C05466=1030.295,97.763,400.155,168.679,44.365,158.305
C05467=1030.301,98.012,400.136,168.682,44.363,158.304
C05468=1030.307,98.261,400.117,168.684,44.361,158.304
C05469=1030.314,98.510,400.099,168.687,44.358,158.304
C05470=1030.319,98.759,400.079,168.688,44.356,158.304
C05471=1030.326,99.008,400.060,168.691,44.354,158.304
C05472=1030.332,99.258,400.041,168.693,44.353,158.304
C05473=1030.338,99.507,400.022,168.696,44.351,158.303
C05474=1030.344,99.756,400.003,168.698,44.349,158.303
C05475=1030.350,100.005,399.984,168.701,44.347,158.303
C05476=1030.356,100.254,399.964,168.704,44.345,158.303
C05477=1030.362,100.504,399.945,168.706,44.343,158.303
C05478=1030.368,100.754,399.926,168.708,44.341,158.303
C05479=1030.375,101.002,399.906,168.710,44.339,158.303
C05480=1030.381,101.252,399.887,168.713,44.337,158.302
C05481=1030.386,101.501,399.868,168.715,44.335,158.302
C05482=1030.393,101.750,399.848,168.718,44.334,158.302
C05483=1030.399,101.999,399.829,168.721,44.332,158.302
C05484=1030.404,102.249,399.810,168.723,44.330,158.302
C05485=1030.410,102.497,399.790,168.725,44.328,158.302
C05486=1030.417,102.746,399.771,168.727,44.326,158.302
C05487=1030.422,102.996,399.752,168.730,44.324,158.301
C05488=1030.428,103.245,399.732,168.733,44.322,158.301
C05489=1030.435,103.494,399.713,168.735,44.320,158.301
C05490=1030.441,103.743,399.693,168.738,44.318,158.301
C05491=1030.447,103.992,399.674,168.740,44.316,158.301
C05492=1030.453,104.242,399.655,168.742,44.315,158.301
C05493=1030.460,104.491,399.635,168.744,44.313,158.301
C05494=1030.465,104.740,399.616,168.747,44.311,158.300
C05495=1030.471,104.989,399.596,168.749,44.308,158.300
C05496=1030.477,105.238,399.577,168.752,44.306,158.300
C05497=1030.483,105.487,399.558,168.755,44.304,158.300
C05498=1030.489,105.736,399.538,168.757,44.303,158.300
C05499=1030.495,105.986,399.519,168.760,44.301,158.300
C05500=1030.502,106.235,399.499,168.761,44.299,158.299
C05501=1030.508,106.484,399.480,168.764,44.297,158.299
C05502=1030.514,106.733,399.460,168.767,44.295,158.299
C05503=1030.520,106.983,399.441,168.769,44.293,158.299
C05504=1030.526,107.231,399.421,168.772,44.291,158.299
C05505=1030.532,107.481,399.402,168.774,44.289,158.299
C05506=1030.538,107.729,399.382,168.777,44.287,158.299
C05507=1030.546,108.015,399.360,168.779,44.285,158.298
C05508=1030.552,108.300,399.338,168.782,44.283,158.298
C05509=1030.560,108.586,399.315,168.785,44.281,158.298
C05510=1030.566,108.871,399.293,168.788,44.278,158.298
C05511=1030.573,109.120,399.274,168.790,44.276,158.298
C05512=1030.579,109.368,399.254,168.793,44.274,158.298
C05513=1030.585,109.619,399.234,168.796,44.272,158.297
C05514=1030.591,109.867,399.214,168.798,44.271,158.297
C05515=1030.597,110.116,399.195,168.801,44.269,158.297
C05516=1030.603,110.365,399.175,168.803,44.267,158.297
C05517=1030.610,110.615,399.156,168.805,44.265,158.297
C05518=1030.616,110.864,399.136,168.807,44.263,158.297
C05519=1030.622,111.113,399.116,168.810,44.261,158.297
C05520=1030.627,111.362,399.097,168.813,44.259,158.296
C05521=1030.633,111.611,399.077,168.815,44.257,158.296
C05522=1030.640,111.861,399.056,168.818,44.255,158.296
C05523=1030.646,112.110,399.037,168.820,44.253,158.296
C05524=1030.652,112.359,399.017,168.823,44.252,158.296
C05525=1030.658,112.608,398.997,168.826,44.250,158.296
C05526=1030.663,112.857,398.978,168.828,44.248,158.296
C05527=1030.670,113.107,398.958,168.830,44.246,158.295
C05528=1030.676,113.356,398.938,168.832,44.244,158.295
C05529=1030.682,113.604,398.918,168.835,44.242,158.295
C05530=1030.688,113.854,398.898,168.838,44.241,158.295
C05531=1030.694,114.103,398.878,168.840,44.239,158.295
C05532=1030.699,114.352,398.858,168.843,44.237,158.295
C05533=1030.705,114.601,398.838,168.845,44.235,158.295
C05534=1030.711,114.850,398.818,168.847,44.234,158.294
C05535=1030.717,115.099,398.798,168.850,44.232,158.294
C05536=1030.724,115.349,398.778,168.852,44.230,158.294
C05537=1030.729,115.598,398.758,168.855,44.228,158.294
C05538=1030.735,115.847,398.738,168.858,44.227,158.294
C05539=1030.741,116.096,398.718,168.860,44.225,158.294
C05540=1030.748,116.345,398.697,168.863,44.223,158.294
C05541=1030.754,116.594,398.677,168.865,44.221,158.294
C05542=1030.759,116.843,398.657,168.867,44.219,158.293
C05543=1030.765,117.092,398.637,168.870,44.217,158.293
C05544=1030.771,117.342,398.617,168.872,44.215,158.293
C05545=1030.777,117.590,398.597,168.875,44.213,158.293
C05546=1030.783,117.840,398.577,168.878,44.212,158.293
C05547=1030.788,118.089,398.557,168.880,44.210,158.293
C05548=1030.795,118.338,398.536,168.883,44.208,158.293
C05549=1030.801,118.587,398.516,168.885,44.206,158.293
C05550=1030.807,118.836,398.497,168.888,44.204,158.293
C05551=1030.813,119.086,398.476,168.889,44.203,158.292
C05552=1030.819,119.335,398.456,168.892,44.201,158.292
C05553=1030.825,119.584,398.436,168.895,44.199,158.292
C05554=1030.831,119.833,398.415,168.897,44.197,158.292
C05555=1030.837,120.082,398.395,168.900,44.195,158.292
C05556=1030.843,120.331,398.375,168.903,44.194,158.292
C05557=1030.849,120.581,398.355,168.905,44.192,158.292
C05558=1030.855,120.829,398.335,168.908,44.190,158.291
C05559=1030.861,121.078,398.315,168.910,44.188,158.291
C05560=1030.867,121.328,398.294,168.913,44.186,158.291
C05561=1030.873,121.577,398.274,168.916,44.184,158.291
C05562=1030.879,121.826,398.254,168.918,44.182,158.291
C05563=1030.886,122.075,398.233,168.920,44.181,158.291
C05564=1030.892,122.324,398.213,168.922,44.179,158.291
C05565=1030.897,122.573,398.193,168.925,44.177,158.290
C05566=1030.904,122.822,398.172,168.927,44.175,158.290
C05567=1030.910,123.071,398.152,168.930,44.173,158.290
C05568=1030.916,123.320,398.132,168.933,44.172,158.290
C05569=1030.922,123.569,398.111,168.935,44.170,158.290
C05570=1030.928,123.818,398.091,168.938,44.168,158.290
C05571=1030.935,124.104,398.067,168.940,44.165,158.290
C05572=1030.942,124.388,398.045,168.944,44.163,158.290
C05573=1030.949,124.673,398.021,168.947,44.161,158.289
C05574=1030.956,124.959,397.997,168.950,44.159,158.289
C05575=1030.962,125.208,397.977,168.953,44.157,158.289
C05576=1030.968,125.457,397.957,168.955,44.156,158.289
C05577=1030.974,125.706,397.937,168.958,44.154,158.289
C05578=1030.980,125.955,397.917,168.960,44.152,158.289
C05579=1030.986,126.205,397.896,168.962,44.150,158.289
C05580=1030.993,126.453,397.876,168.965,44.148,158.288
C05581=1030.999,126.702,397.855,168.967,44.146,158.288
C05582=1031.004,126.951,397.835,168.970,44.144,158.288
C05583=1031.011,127.201,397.814,168.973,44.142,158.288
C05584=1031.017,127.450,397.794,168.975,44.141,158.288
C05585=1031.024,127.699,397.773,168.978,44.139,158.288
C05586=1031.029,127.948,397.753,168.980,44.137,158.288
C05587=1031.036,128.197,397.733,168.983,44.135,158.287
C05588=1031.042,128.446,397.713,168.985,44.133,158.287
C05589=1031.049,128.695,397.692,168.988,44.131,158.287
C05590=1031.054,128.944,397.671,168.991,44.129,158.287
C05591=1031.060,129.194,397.651,168.993,44.128,158.287
C05592=1031.066,129.442,397.631,168.996,44.126,158.287
C05593=1031.073,129.692,397.609,168.999,44.124,158.287
C05594=1031.079,129.940,397.589,169.001,44.122,158.287
C05595=1031.085,130.190,397.569,169.004,44.120,158.286
C05596=1031.092,130.438,397.548,169.006,44.118,158.286
C05597=1031.097,130.688,397.527,169.009,44.116,158.286
C05598=1031.103,130.937,397.507,169.012,44.115,158.286
C05599=1031.110,131.186,397.486,169.014,44.113,158.286
C05600=1031.115,131.435,397.465,169.017,44.111,158.286
C05601=1031.122,131.684,397.444,169.020,44.110,158.286
C05602=1031.127,131.933,397.423,169.022,44.108,158.286
C05603=1031.134,132.183,397.403,169.025,44.106,158.285
C05604=1031.139,132.431,397.382,169.027,44.104,158.285
C05605=1031.146,132.681,397.362,169.030,44.102,158.285
C05606=1031.151,132.929,397.340,169.033,44.101,158.285
C05607=1031.157,133.179,397.319,169.035,44.099,158.285
C05608=1031.163,133.427,397.299,169.038,44.097,158.285
C05609=1031.169,133.677,397.278,169.041,44.095,158.285
C05610=1031.176,133.925,397.257,169.043,44.093,158.285
C05611=1031.181,134.175,397.236,169.046,44.091,158.284
C05612=1031.187,134.423,397.215,169.049,44.090,158.284
C05613=1031.194,134.673,397.195,169.051,44.088,158.284
C05614=1031.199,134.922,397.173,169.054,44.086,158.284
C05615=1031.206,135.170,397.152,169.056,44.084,158.284
C05616=1031.211,135.420,397.132,169.059,44.082,158.284
C05617=1031.217,135.669,397.110,169.062,44.081,158.284
C05618=1031.224,135.918,397.090,169.064,44.079,158.284
C05619=1031.230,136.167,397.068,169.067,44.077,158.284
C05620=1031.236,136.416,397.048,169.069,44.075,158.283
C05621=1031.242,136.665,397.027,169.072,44.074,158.283
C05622=1031.248,136.914,397.005,169.075,44.072,158.283
C05623=1031.255,137.163,396.985,169.077,44.070,158.283
C05624=1031.260,137.412,396.964,169.080,44.069,158.283
C05625=1031.266,137.661,396.942,169.083,44.067,158.283
C05626=1031.272,137.910,396.922,169.085,44.065,158.283
C05627=1031.278,138.159,396.900,169.088,44.064,158.283
C05628=1031.284,138.408,396.879,169.091,44.062,158.283
C05629=1031.290,138.658,396.858,169.093,44.060,158.282
C05630=1031.297,138.906,396.837,169.096,44.058,158.282
C05631=1031.302,139.155,396.816,169.099,44.057,158.282
C05632=1031.308,139.405,396.795,169.101,44.055,158.282
C05633=1031.314,139.654,396.773,169.104,44.053,158.282
C05634=1031.320,139.902,396.752,169.106,44.051,158.282
C05635=1031.327,140.187,396.728,169.110,44.049,158.282
C05636=1031.334,140.473,396.704,169.113,44.048,158.282
C05637=1031.341,140.758,396.679,169.115,44.046,158.282
C05638=1031.347,141.042,396.655,169.119,44.044,158.282
C05639=1031.354,141.291,396.633,169.122,44.042,158.281
C05640=1031.360,141.541,396.613,169.124,44.040,158.281
C05641=1031.365,141.789,396.591,169.127,44.039,158.281
C05642=1031.371,142.039,396.570,169.130,44.037,158.281
C05643=1031.378,142.287,396.549,169.132,44.035,158.281
C05644=1031.384,142.536,396.527,169.135,44.033,158.281
C05645=1031.390,142.785,396.506,169.138,44.032,158.281
C05646=1031.396,143.034,396.484,169.140,44.030,158.281
C05647=1031.401,143.283,396.463,169.143,44.028,158.281
C05648=1031.407,143.533,396.442,169.146,44.027,158.281
C05649=1031.414,143.782,396.420,169.148,44.025,158.280
C05650=1031.420,144.030,396.400,169.151,44.023,158.280
C05651=1031.426,144.279,396.378,169.153,44.021,158.280
C05652=1031.432,144.528,396.356,169.156,44.020,158.280
C05653=1031.438,144.778,396.335,169.159,44.018,158.280
C05654=1031.444,145.026,396.313,169.161,44.016,158.280
C05655=1031.450,145.275,396.292,169.165,44.015,158.280
C05656=1031.456,145.525,396.270,169.168,44.013,158.280
C05657=1031.462,145.773,396.249,169.170,44.011,158.280
C05658=1031.469,146.022,396.228,169.173,44.009,158.279
C05659=1031.475,146.271,396.206,169.176,44.008,158.279
C05660=1031.481,146.520,396.185,169.178,44.006,158.279
C05661=1031.487,146.769,396.163,169.181,44.004,158.279
C05662=1031.493,147.018,396.142,169.184,44.003,158.279
C05663=1031.499,147.267,396.120,169.186,44.001,158.279
C05664=1031.505,147.517,396.098,169.189,43.999,158.279
C05665=1031.511,147.765,396.077,169.192,43.998,158.279
C05666=1031.517,148.014,396.055,169.194,43.996,158.279
C05667=1031.522,148.264,396.033,169.197,43.994,158.279
C05668=1031.528,148.513,396.012,169.200,43.993,158.279
C05669=1031.534,148.761,395.990,169.202,43.991,158.278
C05670=1031.540,149.011,395.969,169.205,43.990,158.278
C05671=1031.546,149.260,395.947,169.209,43.987,158.278
C05672=1031.553,149.508,395.925,169.212,43.986,158.278
C05673=1031.558,149.757,395.903,169.214,43.984,158.278
C05674=1031.565,150.006,395.882,169.217,43.982,158.278
C05675=1031.571,150.255,395.860,169.220,43.981,158.278
C05676=1031.576,150.505,395.838,169.222,43.979,158.278
C05677=1031.582,150.753,395.816,169.225,43.977,158.278
C05678=1031.588,151.002,395.794,169.228,43.976,158.278
C05679=1031.594,151.251,395.773,169.230,43.974,158.278
C05680=1031.600,151.500,395.751,169.233,43.973,158.278
C05681=1031.607,151.750,395.729,169.236,43.971,158.277
C05682=1031.613,151.998,395.707,169.238,43.969,158.277
C05683=1031.618,152.247,395.685,169.242,43.968,158.277
C05684=1031.624,152.496,395.664,169.245,43.966,158.277
C05685=1031.630,152.745,395.642,169.248,43.965,158.277
C05686=1031.637,152.994,395.620,169.250,43.963,158.277
C05687=1031.643,153.243,395.598,169.253,43.962,158.277
C05688=1031.649,153.492,395.576,169.256,43.960,158.277
C05689=1031.655,153.740,395.554,169.258,43.958,158.277
C05690=1031.660,153.990,395.532,169.261,43.957,158.277
C05691=1031.666,154.239,395.510,169.264,43.955,158.277
C05692=1031.673,154.488,395.488,169.266,43.954,158.277
C05693=1031.678,154.737,395.466,169.270,43.952,158.276
C05694=1031.685,154.986,395.444,169.273,43.950,158.276
C05695=1031.690,155.234,395.422,169.275,43.948,158.276
C05696=1031.697,155.483,395.401,169.278,43.947,158.276
C05697=1031.702,155.732,395.378,169.281,43.945,158.276
C05698=1031.708,155.982,395.356,169.284,43.944,158.276
C05699=1031.715,156.266,395.330,169.287,43.942,158.276
C05700=1031.722,156.551,395.305,169.290,43.940,158.276
C05701=1031.730,156.835,395.280,169.293,43.938,158.276
C05702=1031.736,157.120,395.255,169.296,43.937,158.276
C05703=1031.742,157.369,395.232,169.300,43.935,158.276
C05704=1031.748,157.618,395.211,169.303,43.934,158.276
C05705=1031.754,157.867,395.188,169.305,43.932,158.276
C05706=1031.761,158.116,395.167,169.308,43.930,158.276
C05707=1031.766,158.364,395.144,169.311,43.929,158.275
C05708=1031.772,158.614,395.123,169.314,43.927,158.275
C05709=1031.778,158.862,395.100,169.316,43.925,158.275
C05710=1031.784,159.112,395.078,169.320,43.923,158.275
C05711=1031.790,159.360,395.056,169.323,43.922,158.275
C05712=1031.796,159.609,395.034,169.325,43.920,158.275
C05713=1031.802,159.858,395.011,169.328,43.919,158.275
C05714=1031.808,160.107,394.988,169.331,43.918,158.275
C05715=1031.814,160.356,394.966,169.333,43.916,158.275
C05716=1031.820,160.605,394.943,169.336,43.915,158.275
C05717=1031.826,160.854,394.921,169.339,43.913,158.275
C05718=1031.831,161.104,394.898,169.342,43.912,158.275
C05719=1031.837,161.352,394.876,169.345,43.910,158.275
C05720=1031.843,161.601,394.853,169.348,43.909,158.275
C05721=1031.848,161.849,394.830,169.351,43.908,158.275
C05722=1031.854,162.099,394.808,169.354,43.906,158.275
C05723=1031.860,162.348,394.786,169.357,43.905,158.275
C05724=1031.866,162.596,394.763,169.359,43.903,158.275
C05725=1031.872,162.845,394.740,169.362,43.902,158.275
C05726=1031.877,163.094,394.717,169.365,43.900,158.274
C05727=1031.884,163.343,394.695,169.368,43.899,158.274
C05728=1031.889,163.592,394.672,169.371,43.898,158.275
C05729=1031.895,163.841,394.649,169.374,43.896,158.274
C05730=1031.901,164.090,394.627,169.377,43.895,158.274
C05731=1031.907,164.339,394.604,169.380,43.893,158.274
C05732=1031.913,164.588,394.581,169.382,43.892,158.274
C05733=1031.918,164.837,394.559,169.385,43.890,158.274
C05734=1031.924,165.086,394.536,169.388,43.889,158.274
C05735=1031.931,165.335,394.514,169.392,43.888,158.274
C05736=1031.936,165.583,394.491,169.395,43.886,158.274
C05737=1031.942,165.832,394.468,169.397,43.884,158.274
C05738=1031.948,166.081,394.445,169.400,43.883,158.274
C05739=1031.954,166.330,394.423,169.403,43.882,158.274
C05740=1031.960,166.579,394.400,169.405,43.880,158.274
C05741=1031.966,166.828,394.377,169.409,43.879,158.274
C05742=1031.971,167.077,394.354,169.412,43.878,158.274
C05743=1031.978,167.325,394.331,169.415,43.876,158.274
C05744=1031.983,167.575,394.309,169.417,43.874,158.274
C05745=1031.989,167.824,394.286,169.420,43.873,158.274
C05746=1031.995,168.072,394.263,169.424,43.872,158.274
C05747=1032.001,168.321,394.241,169.427,43.870,158.274
C05748=1032.007,168.570,394.218,169.429,43.869,158.274
C05749=1032.013,168.819,394.195,169.432,43.867,158.274
C05750=1032.018,169.068,394.172,169.435,43.866,158.274
C05751=1032.025,169.317,394.149,169.439,43.864,158.274
C05752=1032.031,169.566,394.126,169.442,43.863,158.274
C05753=1032.037,169.814,394.103,169.444,43.862,158.274
C05754=1032.043,170.063,394.080,169.447,43.861,158.274
C05755=1032.049,170.312,394.057,169.450,43.859,158.273
C05756=1032.055,170.561,394.034,169.454,43.857,158.273
C05757=1032.061,170.809,394.012,169.456,43.856,158.273
C05758=1032.067,171.058,393.989,169.459,43.855,158.273
C05759=1032.073,171.308,393.965,169.462,43.853,158.273
C05760=1032.079,171.557,393.942,169.466,43.852,158.273
C05761=1032.085,171.805,393.920,169.468,43.850,158.273
C05762=1032.091,172.054,393.897,169.471,43.849,158.273
C05763=1032.098,172.338,393.871,169.475,43.847,158.273
C05764=1032.104,172.623,393.844,169.479,43.846,158.273
C05765=1032.111,172.907,393.818,169.481,43.844,158.273
C05766=1032.119,173.191,393.792,169.485,43.842,158.273
C05767=1032.124,173.439,393.769,169.488,43.841,158.273
C05768=1032.130,173.688,393.746,169.492,43.839,158.273
C05769=1032.136,173.938,393.722,169.494,43.838,158.273
C05770=1032.143,174.187,393.700,169.497,43.837,158.273
C05771=1032.149,174.435,393.676,169.500,43.835,158.273
C05772=1032.155,174.684,393.653,169.504,43.833,158.273
C05773=1032.160,174.933,393.630,169.506,43.832,158.273
C05774=1032.167,175.182,393.607,169.509,43.831,158.273
C05775=1032.173,175.431,393.585,169.513,43.830,158.273
C05776=1032.179,175.679,393.561,169.516,43.828,158.273
C05777=1032.185,175.928,393.538,169.519,43.826,158.273
C05778=1032.191,176.178,393.515,169.522,43.825,158.273
C05779=1032.197,176.426,393.491,169.525,43.824,158.273
C05780=1032.203,176.675,393.468,169.528,43.822,158.273
C05781=1032.210,176.924,393.446,169.531,43.821,158.273
C05782=1032.216,177.173,393.423,169.534,43.819,158.273
C05783=1032.222,177.421,393.399,169.537,43.818,158.273
C05784=1032.228,177.670,393.376,169.540,43.817,158.273
C05785=1032.234,177.920,393.353,169.544,43.815,158.273
C05786=1032.241,178.168,393.330,169.547,43.814,158.273
C05787=1032.247,178.417,393.307,169.549,43.812,158.273
C05788=1032.253,178.666,393.283,169.553,43.811,158.273
C05789=1032.259,178.914,393.260,169.556,43.810,158.273
C05790=1032.265,179.163,393.237,169.559,43.808,158.272
C05791=1032.271,179.412,393.213,169.562,43.806,158.273
C05792=1032.278,179.661,393.190,169.565,43.805,158.273
C05793=1032.284,179.909,393.167,169.569,43.804,158.273
C05794=1032.290,180.159,393.143,169.572,43.803,158.273
C05795=1032.296,180.408,393.120,169.574,43.801,158.272
C05796=1032.302,180.656,393.097,169.578,43.799,158.272
C05797=1032.308,180.906,393.073,169.581,43.798,158.272
C05798=1032.315,181.154,393.050,169.584,43.797,158.272
C05799=1032.321,181.403,393.027,169.588,43.796,158.272
C05800=1032.327,181.651,393.003,169.590,43.794,158.272
C05801=1032.333,181.900,392.980,169.594,43.792,158.272
C05802=1032.340,182.149,392.956,169.597,43.791,158.272
C05803=1032.345,182.398,392.934,169.600,43.790,158.272
C05804=1032.352,182.647,392.909,169.604,43.788,158.272
C05805=1032.359,182.896,392.887,169.606,43.787,158.272
C05806=1032.364,183.145,392.863,169.610,43.785,158.272
C05807=1032.370,183.393,392.839,169.613,43.784,158.272
C05808=1032.376,183.642,392.816,169.616,43.783,158.272
C05809=1032.381,183.891,392.792,169.620,43.782,158.272
C05810=1032.388,184.140,392.768,169.623,43.781,158.272
C05811=1032.393,184.388,392.743,169.625,43.780,158.272
C05812=1032.400,184.638,392.720,169.628,43.778,158.272
C05813=1032.406,184.886,392.696,169.632,43.777,158.272
C05814=1032.411,185.135,392.672,169.635,43.776,158.272
C05815=1032.418,185.384,392.648,169.638,43.775,158.273
C05816=1032.423,185.632,392.624,169.642,43.774,158.273
C05817=1032.429,185.881,392.600,169.645,43.773,158.273
C05818=1032.435,186.131,392.576,169.647,43.771,158.273
C05819=1032.441,186.379,392.553,169.651,43.770,158.273
C05820=1032.447,186.628,392.528,169.654,43.769,158.273
C05821=1032.453,186.876,392.504,169.658,43.768,158.273
C05822=1032.459,187.125,392.481,169.661,43.767,158.273
C05823=1032.465,187.374,392.456,169.664,43.766,158.273
C05824=1032.471,187.622,392.432,169.668,43.764,158.273
C05825=1032.477,187.872,392.408,169.670,43.763,158.273
C05826=1032.482,188.120,392.385,169.673,43.762,158.273
C05827=1032.489,188.404,392.357,169.677,43.760,158.273
C05828=1032.496,188.687,392.329,169.681,43.759,158.273
C05829=1032.502,188.972,392.302,169.685,43.758,158.273
C05830=1032.510,189.256,392.274,169.689,43.757,158.273
C05831=1032.516,189.504,392.251,169.692,43.756,158.273
C05832=1032.521,189.753,392.226,169.695,43.754,158.273
C05833=1032.528,190.002,392.202,169.698,43.753,158.273
C05834=1032.533,190.250,392.178,169.701,43.752,158.273
C05835=1032.539,190.499,392.154,169.705,43.751,158.273
C05836=1032.545,190.748,392.130,169.708,43.750,158.273
C05837=1032.551,190.997,392.106,169.712,43.748,158.273
C05838=1032.557,191.246,392.081,169.715,43.747,158.273
C05839=1032.563,191.494,392.058,169.718,43.746,158.273
C05840=1032.570,191.743,392.034,169.721,43.745,158.274
C05841=1032.576,191.991,392.009,169.724,43.744,158.274
C05842=1032.582,192.240,391.985,169.728,43.743,158.274
C05843=1032.588,192.489,391.960,169.731,43.741,158.274
C05844=1032.594,192.738,391.936,169.735,43.740,158.274
C05845=1032.599,192.986,391.912,169.738,43.739,158.274
C05846=1032.606,193.235,391.888,169.742,43.738,158.274
C05847=1032.612,193.485,391.863,169.744,43.737,158.274
C05848=1032.618,193.733,391.840,169.748,43.735,158.274
C05849=1032.624,193.982,391.814,169.751,43.735,158.274
C05850=1032.630,194.230,391.791,169.755,43.733,158.274
C05851=1032.636,194.479,391.766,169.758,43.732,158.274
C05852=1032.643,194.728,391.742,169.761,43.731,158.274
C05853=1032.648,194.977,391.718,169.765,43.730,158.274
C05854=1032.655,195.225,391.693,169.768,43.729,158.274
C05855=1032.660,195.474,391.669,169.772,43.728,158.274
C05856=1032.667,195.723,391.645,169.774,43.726,158.274
C05857=1032.673,195.972,391.620,169.778,43.726,158.274
C05858=1032.679,196.220,391.596,169.781,43.724,158.274
C05859=1032.685,196.469,391.571,169.785,43.723,158.274
C05860=1032.692,196.718,391.547,169.788,43.722,158.274
C05861=1032.697,196.967,391.523,169.792,43.721,158.275
C05862=1032.704,197.215,391.498,169.795,43.720,158.275
C05863=1032.710,197.464,391.473,169.799,43.718,158.275
C05864=1032.716,197.712,391.450,169.803,43.718,158.275
C05865=1032.722,197.961,391.424,169.805,43.716,158.275
C05866=1032.729,198.210,391.400,169.809,43.715,158.275
C05867=1032.735,198.459,391.376,169.812,43.715,158.275
C05868=1032.741,198.707,391.351,169.816,43.713,158.275
C05869=1032.747,198.956,391.327,169.819,43.712,158.275
C05870=1032.754,199.205,391.302,169.823,43.711,158.275
C05871=1032.760,199.454,391.277,169.826,43.710,158.275
C05872=1032.766,199.702,391.254,169.830,43.709,158.275
C05873=1032.772,199.951,391.228,169.832,43.707,158.275
C05874=1032.779,200.200,391.204,169.837,43.707,158.275
C05875=1032.785,200.449,391.179,169.840,43.705,158.275
C05876=1032.790,200.697,391.155,169.843,43.705,158.276
C05877=1032.796,200.946,391.130,169.847,43.703,158.276
C05878=1032.803,201.195,391.105,169.850,43.703,158.276
C05879=1032.809,201.443,391.080,169.854,43.701,158.276
C05880=1032.815,201.691,391.055,169.857,43.701,158.276
C05881=1032.821,201.941,391.031,169.861,43.699,158.276
C05882=1032.827,202.189,391.005,169.864,43.699,158.276
C05883=1032.833,202.439,390.981,169.868,43.697,158.276
C05884=1032.838,202.687,390.956,169.871,43.697,158.276
C05885=1032.845,202.935,390.930,169.875,43.695,158.276
C05886=1032.851,203.184,390.906,169.879,43.695,158.276
C05887=1032.858,203.433,390.881,169.882,43.693,158.276
C05888=1032.864,203.682,390.856,169.886,43.693,158.277
C05889=1032.869,203.930,390.831,169.888,43.692,158.277
C05890=1032.875,204.179,390.806,169.893,43.691,158.277
C05891=1032.901,205.228,390.700,170.230,43.795,158.327
C05892=1032.911,205.577,390.663,170.234,43.794,158.327
C05893=1032.921,205.926,390.626,170.237,43.795,158.327
C05894=1032.930,206.275,390.590,170.241,43.794,158.328
C05895=1032.940,206.624,390.552,170.244,43.794,158.328
C05896=1032.946,206.873,390.525,170.246,43.794,158.328
C05897=1032.953,207.121,390.499,170.249,43.793,158.328
C05898=1032.960,207.370,390.473,170.251,43.793,158.328
C05899=1032.966,207.618,390.447,170.255,43.793,158.329
C05900=1032.973,207.867,390.420,170.257,43.793,158.329
C05901=1032.980,208.116,390.394,170.260,43.793,158.329
C05902=1032.986,208.364,390.367,170.262,43.792,158.329
C05903=1032.994,208.612,390.341,170.264,43.793,158.329
C05904=1032.999,208.861,390.314,170.267,43.792,158.330
C05905=1033.006,209.110,390.288,170.270,43.792,158.330
C05906=1033.014,209.358,390.262,170.273,43.792,158.330
C05907=1033.020,209.606,390.235,170.275,43.792,158.330
C05908=1033.027,209.855,390.208,170.278,43.791,158.330
C05909=1033.034,210.104,390.181,170.280,43.792,158.331
C05910=1033.040,210.352,390.155,170.282,43.791,158.331
C05911=1033.047,210.601,390.128,170.285,43.791,158.331
C05912=1033.054,210.849,390.102,170.287,43.791,158.331
C05913=1033.061,211.097,390.075,170.291,43.790,158.331
C05914=1033.067,211.346,390.048,170.293,43.791,158.331
C05915=1033.074,211.595,390.022,170.296,43.791,158.332
C05916=1033.080,211.843,389.995,170.298,43.790,158.332
C05917=1033.087,212.091,389.968,170.301,43.790,158.332
C05918=1033.093,212.340,389.941,170.303,43.790,158.332
C05919=1033.100,212.588,389.915,170.307,43.790,158.332
C05920=1033.107,212.837,389.887,170.309,43.790,158.333
C05921=1033.113,213.085,389.861,170.311,43.790,158.333
C05922=1033.120,213.334,389.834,170.314,43.789,158.333
C05923=1033.127,213.582,389.807,170.316,43.790,158.333
C05924=1033.134,213.831,389.780,170.319,43.790,158.333
C05925=1033.140,214.079,389.754,170.321,43.789,158.334
C05926=1033.147,214.328,389.726,170.325,43.789,158.334
C05927=1033.154,214.576,389.700,170.327,43.789,158.334
C05928=1033.160,214.825,389.673,170.330,43.789,158.334
C05929=1033.167,215.073,389.646,170.332,43.789,158.334
C05930=1033.173,215.322,389.619,170.335,43.789,158.335
C05931=1033.181,215.570,389.592,170.338,43.789,158.335
C05932=1033.187,215.818,389.565,170.341,43.788,158.335
C05933=1033.194,216.067,389.539,170.343,43.789,158.335
C05934=1033.200,216.316,389.511,170.346,43.788,158.335
C05935=1033.208,216.564,389.484,170.348,43.788,158.336
C05936=1033.214,216.812,389.457,170.351,43.788,158.336
C05937=1033.221,217.061,389.431,170.353,43.788,158.336
C05938=1033.227,217.309,389.403,170.357,43.788,158.336
C05939=1033.235,217.558,389.377,170.359,43.788,158.336
C05940=1033.241,217.806,389.349,170.362,43.788,158.337
C05941=1033.248,218.054,389.323,170.364,43.787,158.337
C05942=1033.254,218.303,389.295,170.367,43.787,158.337
C05943=1033.262,218.552,389.269,170.369,43.787,158.337
C05944=1033.268,218.800,389.241,170.373,43.787,158.337
C05945=1033.275,219.048,389.215,170.375,43.787,158.338
C05946=1033.281,219.297,389.187,170.378,43.787,158.338
C05947=1033.289,219.545,389.161,170.380,43.787,158.338
C05948=1033.297,219.900,389.122,170.384,43.787,158.338
C05949=1033.307,220.255,389.083,170.389,43.787,158.339
C05950=1033.317,220.609,389.043,170.392,43.787,158.339
C05951=1033.326,220.964,389.004,170.396,43.787,158.339
C05952=1033.333,221.213,388.977,170.398,43.786,158.339
C05953=1033.339,221.461,388.950,170.401,43.786,158.340
C05954=1033.346,221.710,388.922,170.404,43.787,158.340
C05955=1033.353,221.958,388.895,170.407,43.786,158.340
C05956=1033.359,222.207,388.868,170.410,43.786,158.340
C05957=1033.366,222.455,388.840,170.412,43.786,158.341
C05958=1033.372,222.703,388.813,170.416,43.786,158.341
C05959=1033.379,222.951,388.785,170.418,43.786,158.341
C05960=1033.386,223.200,388.759,170.421,43.786,158.341
C05961=1033.393,223.449,388.731,170.423,43.786,158.342
C05962=1033.399,223.697,388.703,170.426,43.786,158.342
C05963=1033.406,223.945,388.676,170.428,43.786,158.342
C05964=1033.413,224.194,388.648,170.432,43.786,158.342
C05965=1033.420,224.443,388.622,170.435,43.786,158.343
C05966=1033.426,224.690,388.594,170.437,43.786,158.343
C05967=1033.432,224.939,388.567,170.440,43.786,158.343
C05968=1033.439,225.187,388.539,170.442,43.786,158.343
C05969=1033.446,225.436,388.511,170.445,43.785,158.343
C05970=1033.453,225.684,388.485,170.448,43.786,158.344
C05971=1033.460,225.933,388.457,170.451,43.786,158.344
C05972=1033.466,226.181,388.429,170.454,43.786,158.344
C05973=1033.473,226.430,388.401,170.456,43.785,158.344
C05974=1033.480,226.678,388.374,170.460,43.786,158.344
C05975=1033.486,226.927,388.346,170.462,43.786,158.345
C05976=1033.494,227.175,388.319,170.465,43.785,158.345
C05977=1033.500,227.423,388.291,170.468,43.785,158.345
C05978=1033.507,227.672,388.263,170.470,43.785,158.345
C05979=1033.514,227.920,388.236,170.474,43.786,158.346
C05980=1033.520,228.168,388.208,170.476,43.785,158.346
C05981=1033.527,228.416,388.181,170.479,43.785,158.346
C05982=1033.533,228.665,388.153,170.482,43.785,158.346
C05983=1033.540,228.913,388.125,170.484,43.786,158.347
C05984=1033.547,229.162,388.097,170.488,43.786,158.347
C05985=1033.553,229.410,388.070,170.490,43.786,158.347
C05986=1033.560,229.659,388.042,170.493,43.785,158.347
C05987=1033.567,229.907,388.014,170.496,43.785,158.348
C05988=1033.573,230.155,387.986,170.498,43.786,158.348
C05989=1033.580,230.404,387.959,170.502,43.786,158.348
C05990=1033.587,230.652,387.931,170.504,43.786,158.348
C05991=1033.593,230.901,387.903,170.507,43.786,158.349
C05992=1033.600,231.149,387.875,170.510,43.785,158.349
C05993=1033.607,231.397,387.847,170.513,43.786,158.349
C05994=1033.613,231.646,387.819,170.516,43.786,158.349
C05995=1033.620,231.894,387.791,170.519,43.786,158.350
C05996=1033.626,232.143,387.763,170.521,43.786,158.350
C05997=1033.633,232.390,387.735,170.525,43.786,158.350
C05998=1033.640,232.639,387.707,170.527,43.786,158.350
C05999=1033.646,232.888,387.679,170.530,43.786,158.351
C06000=1033.653,233.136,387.651,170.533,43.786,158.351
C06001=1033.659,233.385,387.623,170.536,43.787,158.351
C06002=1033.666,233.632,387.595,170.539,43.787,158.351
C06003=1033.673,233.881,387.567,170.542,43.786,158.352
C06004=1033.682,234.228,387.527,170.545,43.787,158.352
C06005=1033.691,234.575,387.488,170.550,43.787,158.352
C06006=1033.700,234.923,387.449,170.554,43.786,158.353
C06007=1033.709,235.270,387.410,170.557,43.787,158.353
C06008=1033.716,235.518,387.382,170.561,43.787,158.353
C06009=1033.724,235.767,387.354,170.564,43.787,158.354
C06010=1033.730,236.015,387.326,170.566,43.787,158.354
C06011=1033.737,236.263,387.297,170.569,43.787,158.354
C06012=1033.743,236.512,387.269,170.573,43.787,158.354
C06013=1033.750,236.760,387.241,170.576,43.787,158.355
C06014=1033.757,237.008,387.213,170.578,43.787,158.355
C06015=1033.763,237.257,387.185,170.581,43.787,158.355
C06016=1033.770,237.505,387.156,170.585,43.787,158.356
C06017=1033.777,237.753,387.128,170.587,43.788,158.356
C06018=1033.784,238.002,387.100,170.590,43.788,158.356
C06019=1033.790,238.250,387.071,170.593,43.788,158.356
C06020=1033.797,238.498,387.043,170.596,43.788,158.357
C06021=1033.804,238.747,387.015,170.599,43.788,158.357
C06022=1033.810,238.995,386.986,170.602,43.788,158.357
C06023=1033.817,239.243,386.958,170.605,43.788,158.357
C06024=1033.824,239.491,386.930,170.608,43.788,158.358
C06025=1033.831,239.740,386.902,170.611,43.788,158.358
C06026=1033.837,239.988,386.873,170.614,43.788,158.358
C06027=1033.844,240.237,386.845,170.616,43.789,158.359
C06028=1033.851,240.484,386.817,170.620,43.789,158.359
C06029=1033.857,240.733,386.788,170.623,43.789,158.359
C06030=1033.864,240.981,386.760,170.626,43.789,158.359
C06031=1033.870,241.229,386.731,170.628,43.789,158.360
C06032=1033.878,241.478,386.702,170.632,43.789,158.360
C06033=1033.884,241.726,386.674,170.635,43.789,158.360
C06034=1033.891,241.974,386.645,170.637,43.789,158.360
C06035=1033.897,242.222,386.616,170.641,43.790,158.361
C06036=1033.904,242.470,386.588,170.644,43.790,158.361
C06037=1033.910,242.720,386.559,170.647,43.790,158.361
C06038=1033.917,242.968,386.530,170.649,43.790,158.362
C06039=1033.924,243.216,386.502,170.653,43.791,158.362
C06040=1033.930,243.464,386.472,170.656,43.791,158.362
C06041=1033.937,243.712,386.445,170.658,43.791,158.363
C06042=1033.943,243.961,386.415,170.662,43.791,158.363
C06043=1033.950,244.209,386.387,170.665,43.792,158.363
C06044=1033.957,244.457,386.358,170.668,43.792,158.364
C06045=1033.964,244.705,386.329,170.671,43.792,158.364
C06046=1033.970,244.954,386.301,170.674,43.792,158.364
C06047=1033.976,245.202,386.272,170.677,43.792,158.364
C06048=1033.983,245.451,386.243,170.681,43.793,158.365
C06049=1033.989,245.699,386.214,170.683,43.793,158.365
C06050=1033.996,245.946,386.185,170.686,43.793,158.365
C06051=1034.002,246.195,386.156,170.689,43.793,158.366
C06052=1034.009,246.443,386.127,170.692,43.794,158.366
C06053=1034.015,246.692,386.098,170.695,43.794,158.366
C06054=1034.022,246.940,386.069,170.698,43.794,158.367
C06055=1034.029,247.188,386.040,170.702,43.794,158.367
C06056=1034.035,247.436,386.011,170.704,43.795,158.367
C06057=1034.042,247.684,385.982,170.707,43.795,158.368
C06058=1034.048,247.933,385.953,170.711,43.795,158.368
C06059=1034.054,248.181,385.924,170.714,43.795,158.368
C06060=1034.063,248.522,385.884,170.718,43.795,158.369
C06061=1034.073,248.863,385.844,170.722,43.796,158.369
C06062=1034.082,249.204,385.804,170.726,43.797,158.370
C06063=1034.091,249.546,385.764,170.731,43.797,158.370
C06064=1034.098,249.795,385.735,170.734,43.797,158.370
C06065=1034.104,250.043,385.705,170.737,43.797,158.371
C06066=1034.110,250.290,385.676,170.740,43.797,158.371
C06067=1034.117,250.539,385.646,170.743,43.798,158.371
C06068=1034.124,250.787,385.618,170.746,43.798,158.372
C06069=1034.130,251.035,385.589,170.750,43.798,158.372
C06070=1034.137,251.284,385.559,170.753,43.799,158.372
C06071=1034.144,251.532,385.530,170.755,43.799,158.373
C06072=1034.150,251.779,385.501,170.759,43.799,158.373
C06073=1034.157,252.028,385.471,170.762,43.800,158.373
C06074=1034.164,252.276,385.443,170.765,43.800,158.374
C06075=1034.171,252.525,385.413,170.769,43.800,158.374
C06076=1034.177,252.772,385.384,170.772,43.800,158.374
C06077=1034.184,253.021,385.355,170.774,43.801,158.375
C06078=1034.190,253.269,385.325,170.778,43.801,158.375
C06079=1034.197,253.518,385.296,170.781,43.801,158.375
C06080=1034.205,253.765,385.267,170.784,43.802,158.376
C06081=1034.211,254.014,385.238,170.788,43.802,158.376
C06082=1034.217,254.262,385.209,170.791,43.802,158.376
C06083=1034.224,254.510,385.178,170.794,43.802,158.377
C06084=1034.230,254.758,385.149,170.797,43.803,158.377
C06085=1034.237,255.007,385.120,170.800,43.803,158.377
C06086=1034.245,255.254,385.091,170.803,43.803,158.378
C06087=1034.251,255.503,385.061,170.807,43.803,158.378
C06088=1034.258,255.751,385.032,170.810,43.804,158.378
C06089=1034.265,255.999,385.002,170.813,43.804,158.379
C06090=1034.271,256.247,384.973,170.817,43.804,158.379
C06091=1034.278,256.496,384.943,170.820,43.805,158.379
C06092=1034.285,256.744,384.914,170.822,43.805,158.380
C06093=1034.291,256.993,384.885,170.826,43.805,158.380
C06094=1034.299,257.240,384.855,170.829,43.806,158.380
C06095=1034.306,257.489,384.826,170.832,43.806,158.381
C06096=1034.312,257.736,384.796,170.836,43.806,158.381
C06097=1034.319,257.985,384.767,170.839,43.807,158.381
C06098=1034.325,258.232,384.737,170.843,43.807,158.382
C06099=1034.332,258.481,384.708,170.846,43.807,158.382
C06100=1034.339,258.729,384.678,170.849,43.807,158.382
C06101=1034.346,258.977,384.649,170.853,43.807,158.383
C06102=1034.354,259.226,384.619,170.856,43.808,158.383
C06103=1034.360,259.474,384.590,170.859,43.808,158.383
C06104=1034.367,259.722,384.560,170.862,43.809,158.384
C06105=1034.374,259.969,384.530,170.865,43.809,158.384
C06106=1034.380,260.218,384.501,170.868,43.809,158.384
C06107=1034.388,260.466,384.471,170.872,43.810,158.385
C06108=1034.394,260.715,384.442,170.875,43.810,158.385
C06109=1034.402,260.963,384.412,170.879,43.810,158.386
C06110=1034.408,261.210,384.382,170.882,43.810,158.386
C06111=1034.415,261.459,384.353,170.885,43.811,158.386
C06112=1034.422,261.707,384.323,170.889,43.811,158.387
C06113=1034.428,261.955,384.292,170.892,43.812,158.387
C06114=1034.435,262.203,384.262,170.895,43.812,158.387
C06115=1034.442,262.451,384.233,170.899,43.813,158.388
C06116=1034.451,262.791,384.192,170.903,43.813,158.388
C06117=1034.460,263.131,384.151,170.908,43.813,158.389
C06118=1034.469,263.471,384.110,170.913,43.815,158.389
C06119=1034.478,263.811,384.069,170.917,43.815,158.390
C06120=1034.485,264.059,384.038,170.920,43.815,158.390
C06121=1034.491,264.307,384.008,170.924,43.816,158.391
C06122=1034.498,264.555,383.978,170.927,43.816,158.391
C06123=1034.506,264.803,383.948,170.931,43.816,158.391
C06124=1034.511,265.051,383.918,170.934,43.817,158.392
C06125=1034.519,265.299,383.887,170.938,43.818,158.392
C06126=1034.526,265.547,383.857,170.941,43.818,158.393
C06127=1034.532,265.795,383.827,170.944,43.818,158.393
C06128=1034.538,266.044,383.798,170.948,43.819,158.393
C06129=1034.546,266.292,383.767,170.951,43.819,158.394
C06130=1034.552,266.540,383.738,170.955,43.820,158.394
C06131=1034.559,266.788,383.707,170.958,43.820,158.394
C06132=1034.566,267.036,383.676,170.961,43.821,158.395
C06133=1034.573,267.283,383.646,170.965,43.821,158.395
C06134=1034.579,267.532,383.616,170.968,43.822,158.396
C06135=1034.586,267.780,383.586,170.972,43.822,158.396
C06136=1034.592,268.028,383.555,170.975,43.823,158.396
C06137=1034.599,268.276,383.525,170.978,43.823,158.397
C06138=1034.605,268.525,383.494,170.982,43.824,158.397
C06139=1034.613,268.773,383.464,170.985,43.824,158.398
C06140=1034.620,269.020,383.434,170.989,43.825,158.398
C06141=1034.626,269.268,383.403,170.992,43.825,158.399
C06142=1034.633,269.517,383.373,170.996,43.826,158.399
C06143=1034.640,269.765,383.342,170.999,43.826,158.399
C06144=1034.646,270.013,383.312,171.002,43.827,158.400
C06145=1034.653,270.261,383.281,171.006,43.827,158.400
C06146=1034.660,270.509,383.251,171.009,43.828,158.401
C06147=1034.666,270.757,383.220,171.013,43.829,158.401
C06148=1034.673,271.005,383.190,171.016,43.829,158.401
C06149=1034.680,271.253,383.159,171.020,43.829,158.402
C06150=1034.687,271.501,383.129,171.023,43.830,158.402
C06151=1034.693,271.749,383.098,171.027,43.831,158.403
C06152=1034.700,271.996,383.068,171.030,43.831,158.403
C06153=1034.707,272.245,383.037,171.034,43.832,158.404
C06154=1034.713,272.493,383.006,171.037,43.833,158.404
C06155=1034.720,272.741,382.975,171.041,43.833,158.404
C06156=1034.727,272.989,382.945,171.044,43.833,158.405
C06157=1034.734,273.236,382.914,171.047,43.834,158.405
C06158=1034.740,273.485,382.883,171.051,43.835,158.406
C06159=1034.747,273.733,382.852,171.054,43.835,158.406
C06160=1034.754,273.981,382.822,171.058,43.836,158.407
C06161=1034.761,274.229,382.790,171.061,43.837,158.407
C06162=1034.767,274.477,382.760,171.065,43.837,158.407
C06163=1034.774,274.724,382.729,171.068,43.838,158.408
C06164=1034.780,274.973,382.699,171.073,43.838,158.408
C06165=1034.787,275.221,382.667,171.076,43.839,158.409
C06166=1034.794,275.469,382.637,171.080,43.840,158.409
C06167=1034.801,275.717,382.606,171.083,43.840,158.410
C06168=1034.807,275.965,382.575,171.087,43.841,158.410
C06169=1034.815,276.213,382.544,171.090,43.842,158.411
C06170=1034.822,276.461,382.513,171.094,43.842,158.411
C06171=1034.827,276.709,382.482,171.097,43.843,158.411
C06172=1034.838,277.053,382.439,171.102,43.843,158.412
C06173=1034.847,277.398,382.396,171.108,43.844,158.413
C06174=1034.856,277.742,382.353,171.112,43.845,158.413
C06175=1034.865,278.087,382.310,171.117,43.846,158.414
C06176=1034.873,278.335,382.279,171.122,43.847,158.414
C06177=1034.879,278.583,382.247,171.125,43.848,158.415
C06178=1034.886,278.831,382.216,171.129,43.848,158.415
C06179=1034.892,279.079,382.185,171.132,43.849,158.416
C06180=1034.899,279.327,382.154,171.136,43.850,158.416
C06181=1034.906,279.575,382.122,171.139,43.851,158.417
C06182=1034.913,279.823,382.091,171.143,43.852,158.417
C06183=1034.919,280.071,382.060,171.146,43.852,158.418
C06184=1034.926,280.319,382.028,171.150,43.853,158.418
C06185=1034.933,280.567,381.997,171.154,43.853,158.419
C06186=1034.940,280.814,381.965,171.158,43.854,158.419
C06187=1034.946,281.063,381.935,171.161,43.855,158.420
C06188=1034.953,281.311,381.903,171.165,43.856,158.420
C06189=1034.959,281.559,381.872,171.168,43.856,158.421
C06190=1034.966,281.807,381.840,171.172,43.857,158.421
C06191=1034.973,282.055,381.809,171.175,43.858,158.421
C06192=1034.980,282.302,381.777,171.180,43.859,158.422
C06193=1034.987,282.550,381.747,171.184,43.860,158.423
C06194=1034.994,282.798,381.715,171.187,43.860,158.423
C06195=1035.000,283.046,381.684,171.191,43.861,158.423
C06196=1035.007,283.294,381.652,171.194,43.861,158.424
C06197=1035.014,283.542,381.621,171.199,43.863,158.425
C06198=1035.021,283.790,381.589,171.202,43.863,158.425
C06199=1035.028,284.037,381.557,171.206,43.864,158.425
C06200=1035.034,284.285,381.526,171.209,43.865,158.426
C06201=1035.041,284.533,381.494,171.213,43.866,158.426
C06202=1035.048,284.781,381.463,171.218,43.866,158.427
C06203=1035.055,285.028,381.432,171.221,43.867,158.427
C06204=1035.061,285.276,381.400,171.225,43.868,158.428
C06205=1035.069,285.525,381.368,171.228,43.869,158.428
C06206=1035.076,285.772,381.336,171.232,43.869,158.429
C06207=1035.082,286.020,381.305,171.236,43.870,158.429
C06208=1035.089,286.268,381.273,171.240,43.871,158.430
C06209=1035.096,286.516,381.242,171.243,43.872,158.430
C06210=1035.103,286.764,381.210,171.247,43.872,158.431
C06211=1035.110,287.011,381.178,171.251,43.874,158.432
C06212=1035.116,287.259,381.146,171.255,43.874,158.432
C06213=1035.123,287.508,381.114,171.259,43.875,158.432
C06214=1035.130,287.755,381.082,171.262,43.876,158.433
C06215=1035.137,288.003,381.051,171.266,43.877,158.433
C06216=1035.143,288.251,381.019,171.271,43.878,158.434
C06217=1035.150,288.498,380.987,171.274,43.878,158.435
C06218=1035.156,288.747,380.955,171.278,43.879,158.435
C06219=1035.164,288.995,380.923,171.281,43.880,158.436
C06220=1035.171,289.242,380.891,171.286,43.881,158.436
C06221=1035.178,289.490,380.859,171.290,43.882,158.437
C06222=1035.184,289.738,380.827,171.293,43.883,158.437
C06223=1035.191,289.985,380.795,171.297,43.884,158.438
C06224=1035.198,290.234,380.763,171.301,43.884,158.438
C06225=1035.205,290.481,380.731,171.305,43.886,158.439
C06226=1035.211,290.729,380.699,171.309,43.886,158.439
C06227=1035.218,290.977,380.667,171.312,43.888,158.440
C06228=1035.228,291.334,380.621,171.318,43.888,158.441
C06229=1035.239,291.691,380.575,171.324,43.890,158.441
C06230=1035.248,292.046,380.528,171.330,43.891,158.442
C06231=1035.258,292.403,380.482,171.335,43.892,158.443
C06232=1035.265,292.651,380.450,171.339,43.894,158.444
C06233=1035.271,292.900,380.418,171.343,43.894,158.444
C06234=1035.279,293.147,380.386,171.347,43.895,158.445
C06235=1035.286,293.394,380.353,171.351,43.897,158.445
C06236=1035.292,293.642,380.321,171.355,43.897,158.446
C06237=1035.299,293.890,380.289,171.359,43.898,158.446
C06238=1035.305,294.138,380.256,171.363,43.899,158.447
C06239=1035.312,294.385,380.224,171.367,43.900,158.447
C06240=1035.320,294.633,380.191,171.371,43.901,158.448
C06241=1035.326,294.881,380.159,171.375,43.902,158.449
C06242=1035.333,295.129,380.127,171.379,43.903,158.449
C06243=1035.340,295.377,380.094,171.383,43.904,158.450
C06244=1035.346,295.625,380.061,171.386,43.906,158.450
C06245=1035.353,295.872,380.029,171.391,43.907,158.451
C06246=1035.360,296.119,379.997,171.395,43.907,158.451
C06247=1035.367,296.368,379.963,171.398,43.909,158.452
C06248=1035.373,296.615,379.931,171.403,43.910,158.453
C06249=1035.380,296.863,379.899,171.407,43.911,158.453
C06250=1035.387,297.111,379.865,171.410,43.912,158.454
C06251=1035.393,297.359,379.833,171.415,43.913,158.455
C06252=1035.400,297.606,379.799,171.419,43.914,158.455
C06253=1035.407,297.853,379.767,171.422,43.915,158.456
C06254=1035.414,298.101,379.734,171.427,43.916,158.456
C06255=1035.420,298.349,379.701,171.431,43.917,158.457
C06256=1035.427,298.597,379.668,171.435,43.919,158.457
C06257=1035.434,298.844,379.636,171.439,43.920,158.458
C06258=1035.441,299.093,379.603,171.443,43.921,158.459
C06259=1035.447,299.340,379.570,171.447,43.922,158.459
C06260=1035.454,299.588,379.536,171.452,43.923,158.460
C06261=1035.461,299.835,379.504,171.455,43.924,158.461
C06262=1035.468,300.083,379.471,171.460,43.926,158.461
C06263=1035.474,300.331,379.438,171.464,43.926,158.462
C06264=1035.481,300.578,379.405,171.467,43.927,158.462
C06265=1035.489,300.826,379.372,171.472,43.928,158.463
C06266=1035.495,301.074,379.340,171.476,43.930,158.464
C06267=1035.502,301.322,379.306,171.480,43.931,158.464
C06268=1035.508,301.569,379.273,171.484,43.932,158.465
C06269=1035.516,301.817,379.240,171.488,43.933,158.465
C06270=1035.522,302.064,379.208,171.493,43.934,158.466
C06271=1035.530,302.312,379.174,171.496,43.936,158.467
C06272=1035.536,302.560,379.141,171.501,43.937,158.467
C06273=1035.543,302.808,379.109,171.505,43.938,158.468
C06274=1035.551,303.055,379.075,171.510,43.939,158.469
C06275=1035.557,303.303,379.042,171.513,43.940,158.469
C06276=1035.564,303.551,379.008,171.517,43.941,158.470
C06277=1035.570,303.798,378.976,171.522,43.942,158.470
C06278=1035.578,304.046,378.942,171.526,43.944,158.471
C06279=1035.585,304.293,378.910,171.531,43.945,158.472
C06280=1035.592,304.541,378.876,171.534,43.947,158.472
C06281=1035.599,304.789,378.843,171.539,43.948,158.473
C06282=1035.606,305.036,378.810,171.543,43.949,158.474
C06283=1035.613,305.284,378.777,171.547,43.950,158.474
C06284=1035.623,305.657,378.727,171.554,43.952,158.475
C06285=1035.634,306.031,378.676,171.560,43.953,158.476
C06286=1035.644,306.404,378.626,171.567,43.955,158.477
C06287=1035.655,306.778,378.576,171.573,43.957,158.478
C06288=1035.662,307.026,378.542,171.577,43.959,158.479
C06289=1035.669,307.273,378.509,171.582,43.960,158.480
C06290=1035.676,307.521,378.476,171.585,43.961,158.480
C06291=1035.684,307.768,378.442,171.590,43.962,158.481
C06292=1035.690,308.015,378.409,171.594,43.964,158.482
C06293=1035.697,308.263,378.375,171.599,43.965,158.482
C06294=1035.704,308.511,378.342,171.603,43.966,158.483
C06295=1035.712,308.759,378.309,171.607,43.967,158.484
C06296=1035.719,309.006,378.275,171.612,43.968,158.484
C06297=1035.726,309.253,378.242,171.616,43.970,158.485
C06298=1035.733,309.502,378.208,171.621,43.971,158.486
C06299=1035.740,309.749,378.175,171.624,43.972,158.486
C06300=1035.748,309.997,378.141,171.629,43.973,158.487
C06301=1035.755,310.244,378.108,171.634,43.975,158.488
C06302=1035.762,310.491,378.074,171.638,43.976,158.488
C06303=1035.769,310.739,378.040,171.643,43.977,158.489
C06304=1035.776,310.987,378.007,171.646,43.978,158.490
C06305=1035.783,311.235,377.973,171.651,43.980,158.490
C06306=1035.791,311.482,377.940,171.656,43.981,158.491
C06307=1035.798,311.730,377.906,171.660,43.982,158.492
C06308=1035.804,311.977,377.872,171.665,43.984,158.492
C06309=1035.811,312.225,377.838,171.669,43.985,158.493
C06310=1035.819,312.472,377.804,171.673,43.987,158.494
C06311=1035.825,312.720,377.769,171.677,43.989,158.495
C06312=1035.833,312.968,377.736,171.682,43.990,158.495
C06313=1035.838,313.215,377.702,171.686,43.992,158.496
C06314=1035.846,313.462,377.668,171.691,43.993,158.497
C06315=1035.853,313.710,377.633,171.696,43.994,158.498
C06316=1035.860,313.958,377.599,171.700,43.996,158.498
C06317=1035.867,314.205,377.565,171.705,43.997,158.499
C06318=1035.873,314.453,377.531,171.709,43.999,158.500
C06319=1035.880,314.700,377.496,171.713,44.000,158.500
C06320=1035.887,314.948,377.462,171.718,44.002,158.501
C06321=1035.894,315.195,377.428,171.722,44.003,158.502
C06322=1035.901,315.442,377.394,171.727,44.005,158.503
C06323=1035.908,315.690,377.359,171.731,44.006,158.503
C06324=1035.915,315.937,377.325,171.736,44.008,158.504
C06325=1035.922,316.185,377.290,171.741,44.009,158.505
C06326=1035.929,316.433,377.256,171.745,44.011,158.506
C06327=1035.936,316.680,377.221,171.750,44.012,158.506
C06328=1035.943,316.928,377.187,171.754,44.014,158.507
C06329=1035.950,317.175,377.153,171.758,44.015,158.508
C06330=1035.957,317.423,377.118,171.763,44.017,158.509
C06331=1035.964,317.670,377.084,171.767,44.019,158.509
C06332=1035.971,317.918,377.049,171.772,44.020,158.510
C06333=1035.978,318.165,377.015,171.777,44.021,158.511
C06334=1035.985,318.413,376.981,171.781,44.023,158.512
C06335=1035.992,318.660,376.946,171.786,44.025,158.512
C06336=1035.999,318.908,376.912,171.791,44.027,158.513
C06337=1036.006,319.155,376.877,171.795,44.028,158.514
C06338=1036.013,319.403,376.842,171.800,44.029,158.515
C06339=1036.020,319.650,376.808,171.805,44.031,158.516
C06340=1036.031,320.028,376.755,171.811,44.034,158.517
C06341=1036.042,320.406,376.702,171.819,44.036,158.518
C06342=1036.053,320.784,376.650,171.826,44.039,158.519
C06343=1036.065,321.163,376.596,171.834,44.041,158.520
C06344=1036.071,321.410,376.561,171.838,44.043,158.521
C06345=1036.079,321.658,376.527,171.843,44.044,158.522
C06346=1036.085,321.905,376.492,171.848,44.046,158.523
C06347=1036.093,322.152,376.457,171.853,44.048,158.524
C06348=1036.100,322.400,376.422,171.857,44.050,158.524
C06349=1036.108,322.648,376.387,171.862,44.051,158.525
C06350=1036.114,322.896,376.353,171.867,44.053,158.526
C06351=1036.122,323.143,376.318,171.871,44.054,158.527
C06352=1036.128,323.390,376.283,171.875,44.056,158.528
C06353=1036.137,323.638,376.248,171.880,44.058,158.528
C06354=1036.143,323.885,376.213,171.885,44.059,158.529
C06355=1036.151,324.132,376.179,171.890,44.061,158.530
C06356=1036.158,324.380,376.144,171.895,44.063,158.531
C06357=1036.166,324.627,376.109,171.899,44.065,158.532
C06358=1036.172,324.875,376.074,171.904,44.066,158.532
C06359=1036.180,325.122,376.039,171.909,44.068,158.533
C06360=1036.187,325.370,376.004,171.914,44.069,158.534
C06361=1036.195,325.617,375.969,171.919,44.071,158.535
C06362=1036.202,325.864,375.934,171.923,44.073,158.536
C06363=1036.210,326.112,375.899,171.928,44.074,158.537
C06364=1036.216,326.359,375.864,171.933,44.076,158.537
C06365=1036.225,326.607,375.829,171.938,44.078,158.538
C06366=1036.231,326.854,375.794,171.944,44.080,158.539
C06367=1036.239,327.101,375.759,171.948,44.082,158.540
C06368=1036.246,327.350,375.724,171.953,44.083,158.541
C06369=1036.254,327.596,375.688,171.957,44.085,158.542
C06370=1036.261,327.844,375.653,171.962,44.087,158.542
C06371=1036.269,328.091,375.618,171.967,44.088,158.543
C06372=1036.276,328.339,375.583,171.973,44.090,158.544
C06373=1036.283,328.587,375.548,171.978,44.092,158.545
C06374=1036.290,328.833,375.512,171.983,44.094,158.546
C06375=1036.297,329.081,375.476,171.988,44.096,158.547
C06376=1036.305,329.328,375.441,171.992,44.098,158.548
C06377=1036.313,329.576,375.406,171.997,44.100,158.549
C06378=1036.320,329.823,375.370,172.002,44.101,158.549
C06379=1036.327,330.071,375.334,172.007,44.104,158.550
C06380=1036.334,330.318,375.299,172.012,44.105,158.551
C06381=1036.341,330.565,375.263,172.017,44.107,158.552
C06382=1036.349,330.812,375.227,172.023,44.109,158.553
C06383=1036.355,331.060,375.192,172.028,44.111,158.554
C06384=1036.363,331.307,375.156,172.033,44.113,158.555
C06385=1036.370,331.554,375.121,172.037,44.115,158.556
C06386=1036.378,331.802,375.084,172.042,44.117,158.557
C06387=1036.384,332.049,375.049,172.047,44.119,158.558
C06388=1036.392,332.297,375.013,172.052,44.121,158.558
C06389=1036.400,332.544,374.977,172.057,44.123,158.559
C06390=1036.406,332.791,374.942,172.062,44.125,158.560
C06391=1036.414,333.039,374.906,172.068,44.127,158.561
C06392=1036.421,333.286,374.870,172.073,44.128,158.562
C06393=1036.429,333.533,374.833,172.078,44.131,158.563
C06394=1036.436,333.781,374.798,172.083,44.133,158.564
C06395=1036.443,334.028,374.762,172.088,44.134,158.565
C06396=1036.452,334.328,374.718,172.095,44.137,158.566
C06397=1036.461,334.628,374.675,172.101,44.140,158.567
C06398=1036.470,334.928,374.631,172.106,44.142,158.568
C06399=1036.480,335.228,374.587,172.113,44.144,158.569
C06400=1036.487,335.476,374.551,172.118,44.147,158.570
C06401=1036.494,335.723,374.515,172.123,44.149,158.571
C06402=1036.501,335.970,374.479,172.128,44.151,158.572
C06403=1036.509,336.217,374.442,172.134,44.153,158.573
C06404=1036.516,336.464,374.407,172.139,44.155,158.574
C06405=1036.524,336.712,374.370,172.144,44.157,158.575
C06406=1036.531,336.959,374.334,172.149,44.159,158.576
C06407=1036.538,337.206,374.298,172.154,44.161,158.577
C06408=1036.545,337.454,374.261,172.160,44.163,158.578
C06409=1036.553,337.701,374.225,172.165,44.166,158.579
C06410=1036.561,337.948,374.189,172.170,44.168,158.580
C06411=1036.567,338.195,374.152,172.175,44.170,158.581
C06412=1036.575,338.442,374.116,172.181,44.172,158.582
C06413=1036.583,338.690,374.079,172.186,44.174,158.583
C06414=1036.590,338.937,374.043,172.191,44.177,158.584
C06415=1036.597,339.185,374.006,172.196,44.179,158.585
C06416=1036.605,339.431,373.970,172.203,44.181,158.586
C06417=1036.612,339.679,373.934,172.208,44.183,158.587
C06418=1036.620,339.926,373.897,172.213,44.185,158.588
C06419=1036.627,340.174,373.861,172.218,44.187,158.589
C06420=1036.635,340.421,373.824,172.224,44.190,158.590
C06421=1036.643,340.668,373.787,172.229,44.192,158.591
C06422=1036.651,340.915,373.750,172.234,44.194,158.592
C06423=1036.657,341.162,373.714,172.239,44.196,158.593
C06424=1036.667,341.483,373.666,172.247,44.199,158.594
C06425=1036.676,341.803,373.618,172.254,44.202,158.596
C06426=1036.687,342.124,373.571,172.260,44.205,158.597
C06427=1036.696,342.444,373.523,172.268,44.208,158.598
C06428=1036.703,342.692,373.487,172.273,44.211,158.599
C06429=1036.711,342.939,373.449,172.279,44.213,158.600
C06430=1036.718,343.186,373.413,172.284,44.215,158.601
C06431=1036.726,343.433,373.375,172.289,44.218,158.603
C06432=1036.733,343.680,373.338,172.295,44.220,158.604
C06433=1036.740,343.928,373.302,172.300,44.222,158.605
C06434=1036.748,344.175,373.265,172.306,44.225,158.606
C06435=1036.756,344.422,373.227,172.312,44.227,158.607
C06436=1036.764,344.669,373.190,172.317,44.229,158.608
C06437=1036.771,344.917,373.153,172.322,44.232,158.609
C06438=1036.779,345.163,373.117,172.328,44.234,158.610
C06439=1036.786,345.411,373.079,172.334,44.236,158.611
C06440=1036.794,345.657,373.042,172.339,44.239,158.612
C06441=1036.801,345.904,373.005,172.345,44.241,158.613
C06442=1036.809,346.151,372.968,172.350,44.244,158.614
C06443=1036.816,346.398,372.930,172.356,44.246,158.615
C06444=1036.824,346.646,372.892,172.362,44.248,158.616
C06445=1036.832,346.893,372.855,172.367,44.251,158.618
C06446=1036.839,347.140,372.818,172.373,44.254,158.619
C06447=1036.847,347.387,372.781,172.378,44.256,158.620
C06448=1036.855,347.634,372.743,172.385,44.258,158.621
C06449=1036.862,347.881,372.706,172.390,44.261,158.622
C06450=1036.870,348.128,372.669,172.395,44.263,158.623
C06451=1036.878,348.376,372.631,172.401,44.266,158.624
C06452=1036.889,348.747,372.575,172.410,44.269,158.626
C06453=1036.901,349.115,372.519,172.418,44.274,158.628
C06454=1036.912,349.486,372.463,172.427,44.277,158.629
C06455=1036.923,349.856,372.406,172.435,44.281,158.631
C06456=1036.931,350.104,372.369,172.441,44.284,158.632
C06457=1036.938,350.351,372.331,172.447,44.286,158.633
C06458=1036.946,350.597,372.293,172.453,44.289,158.635
C06459=1036.954,350.844,372.256,172.458,44.292,158.636
C06460=1036.962,351.091,372.217,172.465,44.294,158.637
C06461=1036.969,351.339,372.180,172.470,44.297,158.638
C06462=1036.977,351.586,372.142,172.476,44.299,158.639
C06463=1036.984,351.832,372.104,172.482,44.302,158.640
C06464=1036.992,352.080,372.066,172.488,44.305,158.641
C06465=1037.000,352.327,372.028,172.493,44.307,158.643
C06466=1037.007,352.573,371.991,172.500,44.310,158.644
C06467=1037.016,352.821,371.952,172.505,44.313,158.645
C06468=1037.023,353.068,371.915,172.511,44.316,158.646
C06469=1037.030,353.314,371.877,172.517,44.318,158.648
C06470=1037.039,353.561,371.838,172.523,44.321,158.649
C06471=1037.046,353.809,371.800,172.529,44.324,158.650
C06472=1037.054,354.056,371.762,172.535,44.326,158.651
C06473=1037.062,354.302,371.724,172.540,44.329,158.652
C06474=1037.070,354.549,371.687,172.547,44.332,158.653
C06475=1037.078,354.796,371.648,172.552,44.334,158.655
C06476=1037.085,355.043,371.610,172.559,44.338,158.656
C06477=1037.093,355.290,371.571,172.565,44.340,158.657
C06478=1037.101,355.537,371.534,172.571,44.343,158.658
C06479=1037.109,355.784,371.495,172.577,44.346,158.659
C06480=1037.116,356.031,371.457,172.582,44.349,158.661
C06481=1037.124,356.278,371.418,172.589,44.351,158.662
C06482=1037.132,356.525,371.380,172.594,44.354,158.663
C06483=1037.140,356.772,371.341,172.601,44.357,158.665
C06484=1037.148,357.018,371.303,172.607,44.360,158.666
C06485=1037.156,357.266,371.264,172.613,44.363,158.667
C06486=1037.163,357.512,371.226,172.619,44.366,158.668
C06487=1037.172,357.759,371.188,172.626,44.368,158.670
C06488=1037.179,358.006,371.149,172.631,44.372,158.671
C06489=1037.187,358.253,371.111,172.638,44.374,158.672
C06490=1037.195,358.500,371.072,172.644,44.378,158.673
C06491=1037.203,358.747,371.034,172.650,44.380,158.675
C06492=1037.211,358.994,370.995,172.656,44.383,158.676
C06493=1037.219,359.241,370.955,172.662,44.386,158.677
C06494=1037.226,359.488,370.917,172.668,44.389,158.679
C06495=1037.235,359.735,370.879,172.675,44.392,158.680
C06496=1037.242,359.981,370.840,172.681,44.395,158.681
C06497=1037.251,360.228,370.801,172.687,44.398,158.682
C06498=1037.259,360.475,370.762,172.694,44.401,158.684
C06499=1037.267,360.722,370.724,172.699,44.404,158.685
C06500=1037.274,360.968,370.684,172.706,44.407,158.686
C06501=1037.282,361.216,370.646,172.712,44.410,158.688
C06502=1037.291,361.462,370.606,172.719,44.413,158.689
C06503=1037.298,361.709,370.568,172.725,44.416,158.690
C06504=1037.306,361.956,370.529,172.731,44.419,158.692
C06505=1037.314,362.203,370.489,172.738,44.422,158.693
C06506=1037.322,362.450,370.450,172.745,44.425,158.694
C06507=1037.329,362.696,370.411,172.750,44.429,158.696
C06508=1037.342,363.072,370.351,172.760,44.433,158.698
C06509=1037.354,363.448,370.292,172.770,44.438,158.700
C06510=1037.366,363.825,370.231,172.780,44.443,158.702
C06511=1037.378,364.201,370.172,172.789,44.448,158.704
C06512=1037.386,364.448,370.132,172.796,44.451,158.706
C06513=1037.395,364.694,370.093,172.803,44.454,158.707
C06514=1037.402,364.941,370.053,172.810,44.457,158.708
C06515=1037.411,365.188,370.014,172.815,44.461,158.710
C06516=1037.419,365.435,369.975,172.822,44.464,158.711
C06517=1037.427,365.682,369.935,172.829,44.467,158.712
C06518=1037.434,365.928,369.896,172.835,44.470,158.714
C06519=1037.442,366.175,369.856,172.842,44.474,158.715
C06520=1037.451,366.421,369.817,172.849,44.477,158.717
C06521=1037.458,366.668,369.777,172.855,44.480,158.718
C06522=1037.467,366.915,369.738,172.861,44.483,158.719
C06523=1037.475,367.162,369.698,172.868,44.487,158.721
C06524=1037.483,367.408,369.659,172.875,44.490,158.722
C06525=1037.492,367.654,369.618,172.882,44.493,158.724
C06526=1037.499,367.901,369.579,172.888,44.497,158.725
C06527=1037.508,368.148,369.539,172.895,44.500,158.727
C06528=1037.516,368.396,369.499,172.902,44.503,158.728
C06529=1037.525,368.642,369.460,172.908,44.506,158.730
C06530=1037.532,368.889,369.420,172.915,44.510,158.731
C06531=1037.541,369.135,369.380,172.922,44.513,158.733
C06532=1037.550,369.382,369.340,172.928,44.516,158.734
C06533=1037.557,369.629,369.300,172.935,44.520,158.736
C06534=1037.566,369.874,369.260,172.942,44.523,158.737
C06535=1037.574,370.122,369.220,172.949,44.527,158.739
C06536=1037.582,370.369,369.180,172.956,44.530,158.740
C06537=1037.591,370.615,369.140,172.963,44.533,158.741
C06538=1037.599,370.862,369.100,172.970,44.537,158.743
C06539=1037.607,371.108,369.060,172.976,44.541,158.745
C06540=1037.615,371.354,369.019,172.983,44.545,158.746
C06541=1037.623,371.601,368.980,172.990,44.548,158.748
C06542=1037.632,371.848,368.939,172.997,44.551,158.749
C06543=1037.640,372.095,368.899,173.004,44.555,158.751
C06544=1037.648,372.341,368.858,173.011,44.558,158.752
C06545=1037.656,372.588,368.817,173.018,44.562,158.754
C06546=1037.664,372.833,368.777,173.025,44.566,158.755
C06547=1037.673,373.081,368.737,173.032,44.569,158.757
C06548=1037.681,373.327,368.696,173.039,44.573,158.758
C06549=1037.689,373.574,368.656,173.046,44.577,158.760
C06550=1037.697,373.821,368.615,173.053,44.580,158.762
C06551=1037.706,374.067,368.575,173.060,44.584,158.763
C06552=1037.714,374.313,368.534,173.067,44.587,158.765
C06553=1037.723,374.560,368.493,173.074,44.591,158.766
C06554=1037.731,374.806,368.453,173.081,44.595,158.768
C06555=1037.740,375.052,368.413,173.088,44.598,158.769
C06556=1037.748,375.299,368.372,173.095,44.602,158.771
C06557=1037.756,375.545,368.331,173.103,44.605,158.773
C06558=1037.765,375.792,368.290,173.110,44.610,158.774
C06559=1037.773,376.039,368.249,173.117,44.613,158.776
C06560=1037.782,376.285,368.209,173.124,44.617,158.778
C06561=1037.790,376.532,368.168,173.131,44.620,158.779
C06562=1037.799,376.779,368.127,173.138,44.625,158.781
C06563=1037.807,377.025,368.087,173.145,44.628,158.782
C06564=1037.821,377.421,368.020,173.157,44.634,158.785
C06565=1037.835,377.818,367.955,173.169,44.640,158.788
C06566=1037.849,378.214,367.889,173.181,44.647,158.790
C06567=1037.862,378.611,367.822,173.192,44.653,158.793
C06568=1037.870,378.857,367.782,173.200,44.657,158.795
C06569=1037.879,379.104,367.740,173.207,44.660,158.796
C06570=1037.887,379.350,367.699,173.214,44.665,158.798
C06571=1037.896,379.596,367.658,173.222,44.668,158.800
C06572=1037.904,379.842,367.616,173.230,44.673,158.802
C06573=1037.913,380.089,367.575,173.237,44.676,158.803
C06574=1037.921,380.336,367.533,173.244,44.680,158.805
C06575=1037.930,380.581,367.491,173.252,44.685,158.807
C06576=1037.938,380.828,367.450,173.260,44.688,158.809
C06577=1037.947,381.075,367.409,173.267,44.693,158.810
C06578=1037.956,381.320,367.367,173.274,44.696,158.812
C06579=1037.964,381.567,367.325,173.282,44.700,158.814
C06580=1037.972,381.814,367.284,173.289,44.704,158.815
C06581=1037.981,382.060,367.242,173.297,44.708,158.817
C06582=1037.990,382.306,367.201,173.305,44.713,158.819
C06583=1037.999,382.552,367.159,173.312,44.717,158.821
C06584=1038.008,382.799,367.118,173.320,44.721,158.822
C06585=1038.016,383.045,367.075,173.328,44.725,158.824
C06586=1038.025,383.292,367.034,173.335,44.729,158.826
C06587=1038.033,383.537,366.992,173.343,44.733,158.828
C06588=1038.042,383.784,366.951,173.351,44.738,158.830
C06589=1038.051,384.030,366.909,173.358,44.742,158.831
C06590=1038.060,384.276,366.867,173.367,44.746,158.833
C06591=1038.068,384.522,366.824,173.374,44.750,158.835
C06592=1038.077,384.769,366.782,173.381,44.754,158.837
C06593=1038.086,385.015,366.741,173.390,44.758,158.839
C06594=1038.095,385.262,366.699,173.397,44.762,158.841
C06595=1038.104,385.507,366.656,173.406,44.766,158.842
C06596=1038.113,385.754,366.614,173.413,44.771,158.844
C06597=1038.122,386.000,366.572,173.421,44.775,158.846
C06598=1038.131,386.246,366.530,173.429,44.779,158.848
C06599=1038.140,386.492,366.488,173.437,44.784,158.850
C06600=1038.149,386.739,366.447,173.445,44.788,158.852
C06601=1038.157,386.985,366.404,173.453,44.792,158.854
C06602=1038.166,387.231,366.362,173.461,44.796,158.855
C06603=1038.175,387.477,366.319,173.469,44.801,158.857
C06604=1038.184,387.723,366.278,173.477,44.805,158.859
C06605=1038.193,387.969,366.235,173.485,44.809,158.861
C06606=1038.203,388.216,366.192,173.493,44.814,158.863
C06607=1038.212,388.462,366.150,173.501,44.819,158.865
C06608=1038.220,388.708,366.107,173.509,44.823,158.867
C06609=1038.229,388.954,366.065,173.517,44.827,158.869
C06610=1038.238,389.200,366.022,173.525,44.832,158.871
C06611=1038.247,389.446,365.979,173.533,44.836,158.873
C06612=1038.255,389.692,365.937,173.542,44.841,158.875
C06613=1038.265,389.939,365.894,173.550,44.845,158.877
C06614=1038.274,390.185,365.851,173.558,44.850,158.879
C06615=1038.283,390.431,365.809,173.567,44.854,158.881
C06616=1038.291,390.677,365.766,173.574,44.859,158.883
C06617=1038.301,390.923,365.723,173.583,44.863,158.885
C06618=1038.310,391.169,365.680,173.591,44.868,158.886
C06619=1038.319,391.415,365.637,173.599,44.872,158.888
C06620=1038.327,391.630,365.599,173.606,44.877,158.890
C06621=1038.335,391.846,365.562,173.614,44.881,158.892
C06622=1038.343,392.061,365.524,173.621,44.885,158.894
C06623=1038.350,392.277,365.486,173.629,44.889,158.896
C06624=1038.359,392.492,365.448,173.636,44.893,158.897
C06625=1038.367,392.708,365.410,173.643,44.897,158.899
C06626=1038.374,392.924,365.372,173.651,44.901,158.901
C06627=1038.383,393.138,365.334,173.658,44.906,158.903
C06628=1038.391,393.384,365.291,173.667,44.910,158.905
C06629=1038.401,393.631,365.249,173.676,44.914,158.907
C06630=1038.410,393.876,365.205,173.684,44.920,158.909
C06631=1038.419,394.123,365.162,173.692,44.924,158.911
C06632=1038.429,394.368,365.118,173.701,44.929,158.913
C06633=1038.438,394.615,365.075,173.710,44.934,158.915
C06634=1038.447,394.860,365.031,173.719,44.938,158.917
C06635=1038.457,395.106,364.988,173.727,44.944,158.919
C06636=1038.465,395.352,364.945,173.736,44.949,158.922
C06637=1038.475,395.598,364.901,173.744,44.953,158.924
C06638=1038.484,395.844,364.856,173.753,44.958,158.926
C06639=1038.493,396.090,364.813,173.762,44.963,158.928
C06640=1038.503,396.336,364.770,173.771,44.968,158.930
C06641=1038.512,396.582,364.726,173.779,44.973,158.932
C06642=1038.521,396.828,364.682,173.788,44.978,158.934
C06643=1038.530,397.074,364.638,173.797,44.983,158.937
C06644=1038.539,397.319,364.594,173.806,44.988,158.939
C06645=1038.549,397.566,364.550,173.815,44.993,158.941
C06646=1038.559,397.811,364.507,173.824,44.998,158.943
C06647=1038.568,398.058,364.463,173.833,45.003,158.945
C06648=1038.577,398.303,364.419,173.842,45.008,158.948
C06649=1038.587,398.549,364.374,173.850,45.013,158.950
C06650=1038.596,398.795,364.330,173.860,45.018,158.952
C06651=1038.605,399.041,364.286,173.869,45.023,158.954
C06652=1038.615,399.286,364.243,173.878,45.028,158.957
C06653=1038.624,399.532,364.198,173.887,45.034,158.959
C06654=1038.634,399.778,364.154,173.896,45.038,158.961
C06655=1038.644,400.024,364.110,173.905,45.043,158.963
C06656=1038.653,400.270,364.065,173.914,45.049,158.966
C06657=1038.663,400.515,364.021,173.923,45.054,158.968
C06658=1038.672,400.761,363.977,173.932,45.059,158.970
C06659=1038.682,401.007,363.932,173.941,45.064,158.972
C06660=1038.691,401.253,363.888,173.951,45.069,158.975
C06661=1038.701,401.499,363.843,173.960,45.075,158.977
C06662=1038.711,401.744,363.798,173.969,45.080,158.979
C06663=1038.720,401.990,363.754,173.979,45.085,158.982
C06664=1038.730,402.236,363.709,173.988,45.091,158.984
C06665=1038.739,402.482,363.664,173.997,45.096,158.986
C06666=1038.748,402.728,363.619,174.007,45.101,158.989
C06667=1038.758,402.973,363.575,174.017,45.107,158.991
C06668=1038.768,403.219,363.530,174.026,45.112,158.994
C06669=1038.777,403.464,363.485,174.035,45.118,158.996
C06670=1038.788,403.711,363.440,174.044,45.123,158.998
C06671=1038.797,403.956,363.394,174.055,45.129,159.001
C06672=1038.806,404.202,363.350,174.064,45.134,159.003
C06673=1038.816,404.447,363.305,174.073,45.139,159.006
C06674=1038.825,404.693,363.259,174.082,45.145,159.008
C06675=1038.835,404.939,363.214,174.093,45.151,159.011
C06676=1038.845,405.185,363.169,174.102,45.156,159.013
C06677=1038.855,405.430,363.124,174.111,45.162,159.015
C06678=1038.864,405.676,363.078,174.122,45.167,159.018
C06679=1038.874,405.922,363.033,174.131,45.173,159.020
C06680=1038.883,406.147,362.992,174.140,45.178,159.023
C06681=1038.892,406.373,362.950,174.149,45.183,159.025
C06682=1038.901,406.598,362.908,174.159,45.188,159.027
C06683=1038.910,406.823,362.866,174.168,45.193,159.030
C06684=1038.919,407.048,362.825,174.177,45.199,159.032
C06685=1038.928,407.274,362.783,174.185,45.204,159.034
C06686=1038.937,407.498,362.741,174.194,45.209,159.037
C06687=1038.947,407.725,362.699,174.203,45.215,159.039
C06688=1038.956,407.970,362.654,174.214,45.220,159.041
C06689=1038.967,408.216,362.608,174.223,45.226,159.044
C06690=1038.977,408.461,362.562,174.234,45.231,159.047
C06691=1038.986,408.707,362.517,174.243,45.237,159.049
C06692=1038.996,408.952,362.471,174.254,45.243,159.052
C06693=1039.007,409.198,362.425,174.264,45.249,159.054
C06694=1039.017,409.444,362.379,174.274,45.255,159.057
C06695=1039.027,409.689,362.333,174.284,45.261,159.060
C06696=1039.037,409.935,362.288,174.294,45.266,159.062
C06697=1039.047,410.181,362.242,174.305,45.272,159.065
C06698=1039.057,410.426,362.196,174.315,45.278,159.067
C06699=1039.068,410.671,362.150,174.325,45.284,159.070
C06700=1039.078,410.917,362.104,174.336,45.290,159.073
C06701=1039.088,411.163,362.058,174.346,45.296,159.075
C06702=1039.099,411.408,362.012,174.357,45.302,159.078
C06703=1039.109,411.654,361.965,174.367,45.308,159.081
C06704=1039.119,411.900,361.918,174.377,45.314,159.083
C06705=1039.129,412.144,361.873,174.388,45.320,159.086
C06706=1039.139,412.390,361.826,174.399,45.326,159.089
C06707=1039.150,412.635,361.779,174.408,45.332,159.092
C06708=1039.160,412.881,361.733,174.419,45.338,159.094
C06709=1039.170,413.127,361.686,174.430,45.345,159.097
C06710=1039.180,413.372,361.640,174.441,45.351,159.100
C06711=1039.191,413.617,361.593,174.452,45.357,159.103
C06712=1039.200,413.863,361.546,174.463,45.363,159.106
C06713=1039.211,414.108,361.499,174.472,45.369,159.108
C06714=1039.222,414.354,361.452,174.483,45.375,159.111
C06715=1039.232,414.599,361.405,174.494,45.382,159.114
C06716=1039.242,414.845,361.359,174.505,45.388,159.117
C06717=1039.253,415.090,361.312,174.516,45.394,159.120
C06718=1039.263,415.335,361.265,174.527,45.401,159.123
C06719=1039.273,415.580,361.217,174.538,45.407,159.125
C06720=1039.284,415.825,361.171,174.549,45.413,159.128
C06721=1039.294,416.071,361.124,174.560,45.420,159.131
C06722=1039.305,416.317,361.076,174.571,45.426,159.134
C06723=1039.316,416.561,361.029,174.582,45.433,159.137
C06724=1039.326,416.807,360.982,174.593,45.439,159.140
C06725=1039.336,417.052,360.935,174.605,45.445,159.143
C06726=1039.348,417.298,360.888,174.616,45.452,159.146
C06727=1039.358,417.543,360.841,174.627,45.458,159.149
C06728=1039.368,417.788,360.793,174.638,45.464,159.152
C06729=1039.379,418.034,360.745,174.649,45.471,159.155
C06730=1039.389,418.279,360.698,174.660,45.478,159.158
C06731=1039.400,418.524,360.650,174.672,45.484,159.161
C06732=1039.411,418.770,360.603,174.684,45.491,159.164
C06733=1039.421,419.014,360.555,174.695,45.498,159.167
C06734=1039.432,419.260,360.507,174.706,45.504,159.170
C06735=1039.443,419.505,360.460,174.718,45.511,159.173
C06736=1039.454,419.750,360.411,174.729,45.517,159.176
C06737=1039.464,419.995,360.364,174.741,45.525,159.179
C06738=1039.476,420.241,360.316,174.753,45.531,159.182
C06739=1039.486,420.485,360.268,174.764,45.538,159.185
C06740=1039.496,420.715,360.223,174.776,45.544,159.188
C06741=1039.506,420.944,360.177,174.786,45.551,159.191
C06742=1039.516,421.174,360.132,174.797,45.557,159.194
C06743=1039.527,421.404,360.088,174.809,45.563,159.197
C06744=1039.537,421.633,360.042,174.820,45.570,159.200
C06745=1039.547,421.863,359.997,174.831,45.576,159.203
C06746=1039.557,422.092,359.952,174.842,45.583,159.206
C06747=1039.568,422.321,359.907,174.853,45.589,159.209
C06748=1039.579,422.567,359.859,174.865,45.596,159.212
C06749=1039.590,422.812,359.811,174.877,45.603,159.215
C06750=1039.601,423.057,359.762,174.889,45.610,159.219
C06751=1039.612,423.301,359.714,174.901,45.617,159.222
C06752=1039.623,423.547,359.665,174.913,45.624,159.225
C06753=1039.634,423.792,359.616,174.926,45.631,159.228
C06754=1039.645,424.037,359.568,174.938,45.638,159.232
C06755=1039.656,424.282,359.518,174.950,45.645,159.235
C06756=1039.667,424.527,359.470,174.963,45.652,159.238
C06757=1039.679,424.772,359.421,174.975,45.659,159.242
C06758=1039.690,425.017,359.372,174.987,45.666,159.245
C06759=1039.701,425.262,359.324,175.000,45.674,159.248
C06760=1039.712,425.507,359.274,175.012,45.681,159.252
C06761=1039.723,425.752,359.225,175.025,45.688,159.255
C06762=1039.735,425.997,359.176,175.038,45.695,159.259
C06763=1039.746,426.242,359.127,175.051,45.703,159.262
C06764=1039.757,426.487,359.078,175.062,45.710,159.265
C06765=1039.768,426.731,359.029,175.075,45.717,159.269
C06766=1039.779,426.976,358.980,175.088,45.724,159.272
C06767=1039.791,427.222,358.930,175.101,45.732,159.276
C06768=1039.803,427.466,358.881,175.113,45.739,159.279
C06769=1039.813,427.711,358.832,175.126,45.747,159.283
C06770=1039.826,427.956,358.781,175.139,45.754,159.286
C06771=1039.837,428.201,358.732,175.152,45.762,159.290
C06772=1039.848,428.446,358.683,175.165,45.769,159.293
C06773=1039.860,428.690,358.633,175.179,45.776,159.297
C06774=1039.871,428.936,358.583,175.192,45.784,159.301
C06775=1039.883,429.180,358.533,175.205,45.792,159.304
C06776=1039.894,429.424,358.483,175.218,45.800,159.308
C06777=1039.906,429.670,358.434,175.231,45.807,159.311
C06778=1039.917,429.914,358.383,175.244,45.815,159.315
C06779=1039.929,430.159,358.333,175.258,45.822,159.318
C06780=1039.940,430.403,358.283,175.271,45.830,159.322
C06781=1039.952,430.648,358.233,175.284,45.838,159.326
C06782=1039.963,430.893,358.183,175.299,45.845,159.330
C06783=1039.975,431.138,358.132,175.312,45.853,159.333
C06784=1039.986,431.382,358.082,175.325,45.861,159.337
C06785=1039.999,431.627,358.032,175.339,45.869,159.341
C06786=1040.010,431.872,357.981,175.352,45.876,159.344
C06787=1040.022,432.116,357.932,175.367,45.884,159.348
C06788=1040.034,432.361,357.882,175.380,45.892,159.352
C06789=1040.046,432.605,357.830,175.394,45.900,159.356
C06790=1040.058,432.850,357.780,175.408,45.908,159.359
C06791=1040.069,433.095,357.730,175.422,45.916,159.363
C06792=1040.082,433.339,357.679,175.435,45.924,159.367
C06793=1040.094,433.584,357.628,175.450,45.932,159.371
C06794=1040.106,433.828,357.577,175.464,45.940,159.375
C06795=1040.118,434.072,357.526,175.477,45.948,159.379
C06796=1040.130,434.317,357.476,175.492,45.956,159.383
C06797=1040.142,434.561,357.425,175.507,45.964,159.387
C06798=1040.154,434.806,357.374,175.520,45.972,159.390
C06799=1040.166,435.050,357.323,175.535,45.980,159.394
C06800=1040.185,435.425,357.245,175.557,45.993,159.401
C06801=1040.204,435.799,357.166,175.579,46.005,159.407
C06802=1040.222,436.173,357.087,175.602,46.018,159.413
C06803=1040.241,436.547,357.009,175.624,46.031,159.419
C06804=1040.253,436.791,356.958,175.639,46.039,159.423
C06805=1040.265,437.036,356.905,175.654,46.047,159.427
C06806=1040.278,437.280,356.854,175.669,46.056,159.431
C06807=1040.290,437.525,356.803,175.683,46.064,159.435
C06808=1040.302,437.769,356.751,175.698,46.072,159.440
C06809=1040.315,438.013,356.698,175.713,46.081,159.444
C06810=1040.327,438.258,356.647,175.728,46.089,159.448
C06811=1040.340,438.501,356.595,175.743,46.098,159.452
C06812=1040.353,438.746,356.543,175.758,46.107,159.456
C06813=1040.364,438.990,356.492,175.774,46.115,159.461
C06814=1040.377,439.235,356.439,175.789,46.124,159.465
C06815=1040.389,439.479,356.387,175.804,46.133,159.469
C06816=1040.403,439.723,356.335,175.820,46.141,159.473
C06817=1040.415,439.967,356.283,175.835,46.150,159.478
C06818=1040.428,440.212,356.230,175.850,46.158,159.482
C06819=1040.440,440.455,356.178,175.866,46.167,159.486
C06820=1040.453,440.699,356.125,175.881,46.176,159.491
C06821=1040.465,440.943,356.073,175.897,46.185,159.495
C06822=1040.478,441.188,356.021,175.913,46.194,159.500
C06823=1040.491,441.432,355.967,175.929,46.202,159.504
C06824=1040.503,441.676,355.915,175.944,46.211,159.508
C06825=1040.517,441.919,355.863,175.960,46.220,159.513
C06826=1040.530,442.163,355.809,175.977,46.229,159.517
C06827=1040.543,442.408,355.757,175.992,46.238,159.522
C06828=1040.556,442.651,355.704,176.009,46.247,159.526
C06829=1040.569,442.895,355.651,176.025,46.256,159.531
C06830=1040.582,443.139,355.598,176.041,46.265,159.536
C06831=1040.595,443.384,355.545,176.057,46.274,159.540
C06832=1040.613,443.725,355.470,176.080,46.287,159.546
C06833=1040.631,444.066,355.396,176.103,46.300,159.553
C06834=1040.650,444.407,355.322,176.126,46.312,159.560
C06835=1040.668,444.748,355.247,176.150,46.325,159.566
C06836=1040.683,444.990,355.194,176.166,46.334,159.571
C06837=1040.697,445.234,355.142,176.183,46.343,159.575
C06838=1040.712,445.477,355.090,176.200,46.352,159.580
C06839=1040.727,445.721,355.039,176.217,46.361,159.585
C06840=1040.743,445.964,354.988,176.234,46.369,159.589
C06841=1040.760,446.208,354.938,176.251,46.378,159.594
C06842=1040.778,446.453,354.888,176.268,46.387,159.598
C06843=1040.795,446.696,354.838,176.286,46.395,159.603
C06844=1040.814,446.940,354.789,176.303,46.403,159.607
C06845=1040.833,447.185,354.740,176.320,46.411,159.612
C06846=1040.852,447.429,354.693,176.337,46.419,159.616
C06847=1040.872,447.674,354.644,176.356,46.427,159.621
C06848=1040.893,447.918,354.597,176.373,46.435,159.625
C06849=1040.915,448.162,354.550,176.391,46.443,159.630
C06850=1040.937,448.407,354.504,176.408,46.451,159.634
C06851=1040.959,448.651,354.459,176.426,46.458,159.639
C06852=1040.983,448.896,354.413,176.444,46.465,159.643
C06853=1041.006,449.141,354.368,176.462,46.472,159.647
C06854=1041.030,449.386,354.324,176.480,46.480,159.652
C06855=1041.055,449.632,354.280,176.499,46.487,159.656
C06856=1041.082,449.888,354.235,176.518,46.494,159.660
C06857=1041.109,450.145,354.189,176.538,46.501,159.665
C06858=1041.137,450.401,354.146,176.557,46.509,159.670
C06859=1041.166,450.658,354.102,176.576,46.516,159.674
C06860=1041.194,450.904,354.060,176.595,46.523,159.678
C06861=1041.222,451.150,354.019,176.613,46.529,159.683
C06862=1041.251,451.395,353.978,176.632,46.535,159.687
C06863=1041.281,451.640,353.938,176.651,46.542,159.691
C06864=1040.983,451.687,353.621,176.654,46.619,159.715
C06865=1040.954,451.444,353.661,176.635,46.612,159.710
C06866=1040.925,451.201,353.701,176.616,46.606,159.706
C06867=1040.896,450.957,353.742,176.598,46.600,159.702
C06868=1040.869,450.713,353.783,176.579,46.594,159.698
C06869=1040.841,450.469,353.824,176.561,46.586,159.693
C06870=1040.814,450.225,353.866,176.542,46.580,159.689
C06871=1040.788,449.982,353.909,176.523,46.573,159.685
C06872=1040.763,449.738,353.951,176.505,46.566,159.681
C06873=1040.737,449.493,353.994,176.488,46.559,159.676
C06874=1040.713,449.248,354.039,176.469,46.552,159.672
C06875=1040.689,449.003,354.084,176.450,46.545,159.667
C06876=1040.666,448.758,354.129,176.432,46.538,159.663
C06877=1040.642,448.513,354.174,176.414,46.530,159.659
C06878=1040.620,448.269,354.220,176.397,46.523,159.654
C06879=1040.598,448.024,354.267,176.379,46.515,159.650
C06880=1040.578,447.780,354.314,176.361,46.508,159.646
C06881=1040.557,447.535,354.362,176.344,46.500,159.641
C06882=1040.536,447.290,354.410,176.325,46.492,159.636
C06883=1040.517,447.046,354.457,176.308,46.484,159.632
C06884=1040.498,446.803,354.506,176.291,46.475,159.627
C06885=1040.480,446.558,354.555,176.273,46.467,159.623
C06886=1040.462,446.314,354.605,176.256,46.459,159.618
C06887=1040.445,446.070,354.655,176.239,46.451,159.614
C06888=1040.429,445.827,354.706,176.222,46.442,159.609
C06889=1040.413,445.582,354.757,176.205,46.434,159.605
C06890=1040.398,445.339,354.809,176.188,46.425,159.600
C06891=1040.383,445.096,354.861,176.170,46.416,159.595
C06892=1040.368,444.853,354.914,176.154,46.407,159.591
C06893=1040.355,444.609,354.967,176.138,46.398,159.586
C06894=1040.342,444.366,355.019,176.121,46.389,159.582
C06895=1040.329,444.123,355.073,176.104,46.380,159.577
C06896=1040.316,443.879,355.126,176.088,46.371,159.572
C06897=1040.302,443.635,355.179,176.071,46.362,159.568
C06898=1040.289,443.391,355.233,176.054,46.353,159.563
C06899=1040.276,443.147,355.286,176.038,46.344,159.558
C06900=1040.262,442.904,355.338,176.023,46.335,159.554
C06901=1040.250,442.660,355.391,176.006,46.326,159.549
C06902=1040.237,442.416,355.444,175.990,46.317,159.545
C06903=1040.224,442.172,355.497,175.973,46.308,159.540
C06904=1040.211,441.928,355.550,175.958,46.300,159.536
C06905=1040.198,441.683,355.603,175.942,46.290,159.531
C06906=1040.186,441.440,355.655,175.925,46.282,159.527
C06907=1040.173,441.195,355.708,175.910,46.273,159.522
C06908=1040.160,440.951,355.761,175.894,46.264,159.518
C06909=1040.148,440.707,355.813,175.879,46.256,159.514
C06910=1040.135,440.463,355.866,175.863,46.247,159.509
C06911=1040.122,440.218,355.918,175.847,46.238,159.505
C06912=1040.109,439.975,355.971,175.831,46.230,159.501
C06913=1040.096,439.731,356.023,175.816,46.221,159.496
C06914=1040.084,439.487,356.075,175.800,46.213,159.492
C06915=1040.071,439.242,356.128,175.785,46.204,159.488
C06916=1040.059,438.998,356.179,175.770,46.195,159.483
C06917=1040.047,438.763,356.230,175.755,46.187,159.479
C06918=1040.035,438.529,356.279,175.741,46.179,159.475
C06919=1040.022,438.294,356.329,175.726,46.171,159.471
C06920=1040.011,438.060,356.378,175.711,46.163,159.467
C06921=1039.998,437.824,356.429,175.697,46.155,159.463
C06922=1039.987,437.590,356.478,175.683,46.147,159.459
C06923=1039.975,437.356,356.528,175.668,46.139,159.455
C06924=1039.963,437.121,356.578,175.654,46.131,159.451
C06925=1039.951,436.876,356.629,175.639,46.122,159.447
C06926=1039.938,436.632,356.681,175.624,46.114,159.443
C06927=1039.926,436.388,356.732,175.609,46.106,159.439
C06928=1039.914,436.143,356.784,175.595,46.098,159.435
C06929=1039.901,435.895,356.836,175.580,46.089,159.431
C06930=1039.889,435.647,356.888,175.565,46.081,159.427
C06931=1039.877,435.399,356.940,175.551,46.073,159.423
C06932=1039.864,435.151,356.992,175.536,46.065,159.419
C06933=1039.852,434.907,357.044,175.521,46.057,159.415
C06934=1039.840,434.662,357.094,175.507,46.049,159.411
C06935=1039.828,434.417,357.145,175.492,46.041,159.407
C06936=1039.816,434.173,357.196,175.479,46.032,159.403
C06937=1039.804,433.928,357.247,175.464,46.025,159.399
C06938=1039.791,433.684,357.297,175.450,46.017,159.395
C06939=1039.779,433.439,357.348,175.436,46.009,159.391
C06940=1039.767,433.194,357.399,175.422,46.001,159.387
C06941=1039.756,432.950,357.449,175.408,45.993,159.384
C06942=1039.743,432.706,357.500,175.394,45.985,159.380
C06943=1039.732,432.461,357.551,175.380,45.977,159.376
C06944=1039.719,432.216,357.601,175.366,45.970,159.372
C06945=1039.708,431.972,357.652,175.353,45.962,159.369
C06946=1039.696,431.727,357.702,175.338,45.955,159.365
C06947=1039.684,431.482,357.753,175.325,45.946,159.361
C06948=1039.672,431.238,357.802,175.312,45.939,159.357
C06949=1039.661,430.993,357.853,175.298,45.931,159.354
C06950=1039.649,430.749,357.903,175.285,45.923,159.350
C06951=1039.638,430.504,357.953,175.270,45.916,159.346
C06952=1039.626,430.259,358.003,175.257,45.908,159.342
C06953=1039.614,430.015,358.053,175.244,45.901,159.339
C06954=1039.603,429.770,358.104,175.231,45.893,159.335
C06955=1039.591,429.525,358.153,175.217,45.886,159.332
C06956=1039.580,429.280,358.203,175.204,45.878,159.328
C06957=1039.568,429.036,358.253,175.191,45.870,159.324
C06958=1039.557,428.790,358.303,175.178,45.863,159.321
C06959=1039.545,428.546,358.353,175.165,45.855,159.317
C06960=1039.534,428.301,358.402,175.151,45.848,159.314
C06961=1039.522,428.056,358.452,175.138,45.841,159.310
C06962=1039.511,427.812,358.501,175.125,45.833,159.307
C06963=1039.500,427.567,358.551,175.112,45.826,159.303
C06964=1039.488,427.321,358.600,175.099,45.819,159.300
C06965=1039.476,427.077,358.650,175.087,45.811,159.296
C06966=1039.465,426.832,358.699,175.074,45.804,159.293
C06967=1039.454,426.587,358.749,175.061,45.796,159.289
C06968=1039.443,426.342,358.798,175.048,45.790,159.286
C06969=1039.431,426.097,358.847,175.035,45.782,159.282
C06970=1039.419,425.852,358.896,175.023,45.775,159.279
C06971=1039.408,425.608,358.945,175.010,45.768,159.276
C06972=1039.397,425.363,358.995,174.998,45.761,159.272
C06973=1039.386,425.117,359.043,174.985,45.753,159.269
C06974=1039.375,424.872,359.092,174.973,45.746,159.266
C06975=1039.363,424.628,359.141,174.960,45.740,159.262
C06976=1039.352,424.382,359.189,174.948,45.732,159.259
C06977=1039.342,424.137,359.239,174.936,45.725,159.256
C06978=1039.331,423.893,359.288,174.923,45.718,159.252
C06979=1039.320,423.648,359.336,174.911,45.711,159.249
C06980=1039.309,423.402,359.384,174.898,45.704,159.246
C06981=1039.297,423.158,359.433,174.887,45.697,159.242
C06982=1039.286,422.912,359.482,174.874,45.691,159.239
C06983=1039.275,422.667,359.530,174.862,45.684,159.236
C06984=1039.264,422.422,359.579,174.850,45.677,159.233
C06985=1039.253,422.192,359.624,174.839,45.670,159.230
C06986=1039.243,421.961,359.670,174.828,45.664,159.227
C06987=1039.232,421.731,359.715,174.816,45.658,159.224
C06988=1039.222,421.500,359.759,174.805,45.652,159.221
C06989=1039.213,421.269,359.805,174.794,45.645,159.218
C06990=1039.202,421.039,359.850,174.782,45.638,159.215
C06991=1039.192,420.808,359.896,174.772,45.632,159.212
C06992=1039.181,420.578,359.941,174.761,45.626,159.209
C06993=1039.170,420.332,359.989,174.749,45.619,159.206
C06994=1039.160,420.087,360.037,174.737,45.612,159.203
C06995=1039.149,419.842,360.085,174.726,45.606,159.200
C06996=1039.138,419.597,360.133,174.714,45.599,159.197
C06997=1039.127,419.352,360.181,174.702,45.593,159.194
C06998=1039.117,419.106,360.228,174.691,45.586,159.191
C06999=1039.107,418.862,360.276,174.680,45.579,159.187
C07000=1039.096,418.616,360.324,174.667,45.573,159.184
C07001=1039.085,418.371,360.372,174.656,45.566,159.181
C07002=1039.074,418.125,360.419,174.645,45.559,159.178
C07003=1039.064,417.880,360.467,174.634,45.553,159.175
C07004=1039.053,417.635,360.514,174.622,45.547,159.172
C07005=1039.042,417.389,360.561,174.611,45.540,159.169
C07006=1039.032,417.144,360.609,174.600,45.534,159.167
C07007=1039.021,416.900,360.656,174.589,45.527,159.163
C07008=1039.010,416.654,360.704,174.578,45.521,159.161
C07009=1039.000,416.409,360.751,174.567,45.515,159.158
C07010=1038.989,416.164,360.797,174.556,45.508,159.155
C07011=1038.979,415.918,360.845,174.544,45.502,159.152
C07012=1038.969,415.673,360.892,174.533,45.496,159.149
C07013=1038.958,415.427,360.939,174.522,45.490,159.146
C07014=1038.947,415.182,360.986,174.511,45.484,159.143
C07015=1038.937,414.936,361.033,174.500,45.477,159.140
C07016=1038.927,414.691,361.080,174.489,45.471,159.137
C07017=1038.916,414.446,361.126,174.478,45.465,159.135
C07018=1038.906,414.201,361.174,174.467,45.458,159.132
C07019=1038.896,413.955,361.220,174.456,45.453,159.129
C07020=1038.885,413.710,361.267,174.446,45.447,159.126
C07021=1038.875,413.464,361.314,174.436,45.440,159.124
C07022=1038.865,413.219,361.361,174.425,45.434,159.121
C07023=1038.854,412.974,361.407,174.414,45.428,159.118
C07024=1038.844,412.728,361.454,174.403,45.422,159.115
C07025=1038.833,412.483,361.500,174.392,45.416,159.112
C07026=1038.824,412.238,361.546,174.382,45.410,159.110
C07027=1038.814,411.992,361.593,174.372,45.404,159.107
C07028=1038.803,411.747,361.639,174.361,45.398,159.104
C07029=1038.793,411.501,361.686,174.350,45.392,159.101
C07030=1038.782,411.255,361.732,174.340,45.386,159.099
C07031=1038.772,411.009,361.778,174.329,45.380,159.096
C07032=1038.762,410.764,361.824,174.319,45.374,159.093
C07033=1038.752,410.519,361.870,174.309,45.368,159.091
C07034=1038.742,410.273,361.916,174.298,45.363,159.088
C07035=1038.731,410.027,361.962,174.289,45.357,159.086
C07036=1038.721,409.782,362.008,174.278,45.351,159.083
C07037=1038.711,409.536,362.054,174.267,45.345,159.080
C07038=1038.701,409.291,362.100,174.258,45.339,159.078
C07039=1038.690,409.045,362.145,174.247,45.334,159.075
C07040=1038.681,408.799,362.192,174.237,45.328,159.072
C07041=1038.671,408.554,362.237,174.227,45.322,159.070
C07042=1038.661,408.309,362.283,174.217,45.317,159.067
C07043=1038.651,408.062,362.329,174.207,45.311,159.065
C07044=1038.640,407.817,362.375,174.197,45.305,159.062
C07045=1038.631,407.590,362.417,174.187,45.300,159.060
C07046=1038.622,407.364,362.458,174.178,45.295,159.058
C07047=1038.613,407.137,362.500,174.169,45.289,159.055
C07048=1038.604,406.911,362.543,174.160,45.285,159.053
C07049=1038.595,406.685,362.585,174.151,45.279,159.051
C07050=1038.586,406.458,362.626,174.142,45.274,159.048
C07051=1038.577,406.232,362.668,174.132,45.269,159.046
C07052=1038.568,406.005,362.711,174.123,45.264,159.044
C07053=1038.558,405.760,362.755,174.114,45.258,159.041
C07054=1038.548,405.514,362.800,174.105,45.253,159.039
C07055=1038.539,405.268,362.846,174.094,45.248,159.036
C07056=1038.529,405.023,362.892,174.085,45.241,159.034
C07057=1038.519,404.777,362.936,174.076,45.236,159.031
C07058=1038.509,404.532,362.981,174.065,45.231,159.029
C07059=1038.500,404.285,363.027,174.056,45.225,159.026
C07060=1038.490,404.040,363.072,174.047,45.220,159.024
C07061=1038.480,403.794,363.117,174.036,45.215,159.022
C07062=1038.471,403.549,363.162,174.027,45.209,159.019
C07063=1038.461,403.303,363.207,174.018,45.204,159.017
C07064=1038.452,403.058,363.252,174.009,45.198,159.014
C07065=1038.441,402.811,363.297,173.998,45.193,159.012
C07066=1038.432,402.566,363.342,173.989,45.188,159.010
C07067=1038.422,402.320,363.386,173.980,45.182,159.007
C07068=1038.413,402.074,363.431,173.971,45.177,159.005
C07069=1038.403,401.829,363.475,173.961,45.172,159.003
C07070=1038.393,401.582,363.520,173.951,45.167,159.000
C07071=1038.384,401.337,363.565,173.942,45.162,158.998
C07072=1038.375,401.091,363.610,173.933,45.156,158.996
C07073=1038.365,400.845,363.654,173.924,45.151,158.993
C07074=1038.356,400.600,363.699,173.915,45.146,158.991
C07075=1038.346,400.353,363.743,173.906,45.141,158.989
C07076=1038.336,400.108,363.787,173.896,45.136,158.986
C07077=1038.326,399.862,363.831,173.887,45.131,158.984
C07078=1038.318,399.617,363.875,173.877,45.125,158.982
C07079=1038.308,399.371,363.920,173.869,45.121,158.980
C07080=1038.298,399.125,363.964,173.860,45.116,158.977
C07081=1038.289,398.879,364.008,173.851,45.111,158.975
C07082=1038.280,398.633,364.052,173.842,45.106,158.973
C07083=1038.270,398.387,364.096,173.833,45.101,158.971
C07084=1038.260,398.142,364.140,173.823,45.095,158.968
C07085=1038.251,397.896,364.184,173.814,45.090,158.966
C07086=1038.242,397.650,364.228,173.805,45.085,158.964
C07087=1038.232,397.404,364.272,173.797,45.080,158.962
C07088=1038.223,397.158,364.316,173.788,45.076,158.960
C07089=1038.214,396.912,364.360,173.779,45.071,158.957
C07090=1038.204,396.666,364.404,173.770,45.066,158.955
C07091=1038.195,396.420,364.447,173.761,45.061,158.953
C07092=1038.186,396.174,364.491,173.752,45.056,158.951
C07093=1038.176,395.928,364.535,173.744,45.051,158.949
C07094=1038.168,395.683,364.579,173.735,45.046,158.947
C07095=1038.158,395.437,364.622,173.726,45.042,158.945
C07096=1038.149,395.191,364.665,173.717,45.037,158.943
C07097=1038.140,394.944,364.709,173.709,45.032,158.940
C07098=1038.131,394.699,364.753,173.700,45.028,158.938
C07099=1038.121,394.453,364.796,173.691,45.023,158.936
C07100=1038.112,394.207,364.840,173.683,45.018,158.934
C07101=1038.103,393.960,364.883,173.674,45.013,158.932
C07102=1038.093,393.715,364.927,173.666,45.009,158.930
C07103=1038.084,393.469,364.970,173.657,45.004,158.928
C07104=1038.075,393.223,365.013,173.648,44.999,158.926
C07105=1038.068,393.006,365.051,173.641,44.995,158.924
C07106=1038.059,392.790,365.089,173.633,44.991,158.922
C07107=1038.051,392.573,365.127,173.626,44.987,158.920
C07108=1038.043,392.357,365.165,173.618,44.983,158.919
C07109=1038.035,392.140,365.204,173.611,44.979,158.917
C07110=1038.028,391.924,365.241,173.604,44.975,158.915
C07111=1038.019,391.707,365.279,173.596,44.971,158.913
C07112=1038.011,391.491,365.317,173.589,44.967,158.912
C07113=1038.002,391.245,365.359,173.580,44.962,158.910
C07114=1037.993,390.998,365.403,173.573,44.958,158.908
C07115=1037.984,390.752,365.445,173.564,44.953,158.906
C07116=1037.975,390.506,365.488,173.555,44.949,158.904
C07117=1037.966,390.261,365.531,173.548,44.944,158.902
C07118=1037.957,390.014,365.574,173.539,44.940,158.900
C07119=1037.947,389.768,365.617,173.531,44.935,158.898
C07120=1037.939,389.522,365.660,173.523,44.931,158.896
C07121=1037.930,389.276,365.702,173.514,44.926,158.894
C07122=1037.921,389.030,365.745,173.507,44.922,158.892
C07123=1037.912,388.783,365.787,173.498,44.918,158.890
C07124=1037.903,388.537,365.830,173.490,44.913,158.888
C07125=1037.894,388.291,365.873,173.482,44.908,158.886
C07126=1037.885,388.046,365.915,173.473,44.905,158.884
C07127=1037.877,387.799,365.957,173.466,44.900,158.882
C07128=1037.867,387.553,366.000,173.457,44.896,158.880
C07129=1037.858,387.307,366.041,173.450,44.891,158.878
C07130=1037.849,387.060,366.085,173.441,44.888,158.877
C07131=1037.840,386.814,366.127,173.434,44.883,158.875
C07132=1037.831,386.568,366.169,173.425,44.879,158.873
C07133=1037.822,386.322,366.211,173.417,44.874,158.871
C07134=1037.813,386.076,366.253,173.409,44.870,158.869
C07135=1037.804,385.830,366.295,173.402,44.866,158.867
C07136=1037.796,385.583,366.337,173.393,44.862,158.865
C07137=1037.787,385.337,366.380,173.386,44.858,158.864
C07138=1037.778,385.091,366.421,173.378,44.854,158.862
C07139=1037.769,384.844,366.463,173.370,44.850,158.860
C07140=1037.760,384.598,366.505,173.362,44.845,158.858
C07141=1037.751,384.352,366.548,173.354,44.841,158.856
C07142=1037.742,384.106,366.589,173.347,44.837,158.854
C07143=1037.734,383.860,366.631,173.339,44.833,158.853
C07144=1037.725,383.614,366.673,173.331,44.829,158.851
C07145=1037.716,383.367,366.714,173.324,44.825,158.849
C07146=1037.707,383.121,366.756,173.315,44.821,158.847
C07147=1037.699,382.874,366.798,173.308,44.817,158.845
C07148=1037.690,382.628,366.840,173.300,44.813,158.844
C07149=1037.682,382.382,366.881,173.292,44.809,158.842
C07150=1037.673,382.136,366.923,173.285,44.805,158.840
C07151=1037.664,381.889,366.965,173.277,44.800,158.838
C07152=1037.655,381.643,367.007,173.270,44.796,158.837
C07153=1037.647,381.397,367.047,173.262,44.792,158.835
C07154=1037.639,381.150,367.089,173.255,44.789,158.833
C07155=1037.630,380.904,367.131,173.247,44.785,158.831
C07156=1037.621,380.658,367.173,173.240,44.781,158.830
C07157=1037.613,380.411,367.214,173.231,44.777,158.828
C07158=1037.604,380.165,367.255,173.224,44.773,158.826
C07159=1037.596,379.919,367.297,173.217,44.769,158.825
C07160=1037.588,379.672,367.338,173.210,44.765,158.823
C07161=1037.579,379.425,367.380,173.203,44.761,158.821
C07162=1037.570,379.180,367.421,173.194,44.757,158.819
C07163=1037.562,378.933,367.462,173.187,44.753,158.818
C07164=1037.553,378.687,367.504,173.180,44.750,158.816
C07165=1037.539,378.288,367.570,173.168,44.743,158.813
C07166=1037.525,377.890,367.636,173.156,44.737,158.811
C07167=1037.512,377.492,367.703,173.144,44.731,158.808
C07168=1037.497,377.092,367.769,173.133,44.725,158.805
C07169=1037.489,376.846,367.809,173.125,44.722,158.804
C07170=1037.481,376.599,367.851,173.117,44.718,158.802
C07171=1037.472,376.353,367.892,173.110,44.714,158.800
C07172=1037.464,376.106,367.933,173.103,44.710,158.799
C07173=1037.455,375.860,367.973,173.096,44.707,158.797
C07174=1037.446,375.613,368.014,173.089,44.703,158.796
C07175=1037.438,375.367,368.054,173.082,44.700,158.794
C07176=1037.430,375.121,368.095,173.075,44.696,158.792
C07177=1037.422,374.874,368.136,173.068,44.692,158.791
C07178=1037.413,374.628,368.176,173.060,44.688,158.789
C07179=1037.404,374.381,368.217,173.053,44.685,158.788
C07180=1037.396,374.134,368.258,173.046,44.681,158.786
C07181=1037.388,373.888,368.298,173.039,44.678,158.784
C07182=1037.379,373.641,368.339,173.032,44.674,158.783
C07183=1037.371,373.395,368.379,173.025,44.670,158.781
C07184=1037.363,373.148,368.419,173.018,44.667,158.780
C07185=1037.355,372.902,368.460,173.011,44.664,158.778
C07186=1037.347,372.655,368.501,173.004,44.660,158.777
C07187=1037.338,372.409,368.541,172.997,44.656,158.775
C07188=1037.330,372.162,368.581,172.990,44.653,158.774
C07189=1037.322,371.916,368.622,172.983,44.649,158.772
C07190=1037.313,371.669,368.663,172.976,44.646,158.771
C07191=1037.305,371.422,368.702,172.969,44.643,158.769
C07192=1037.297,371.176,368.742,172.962,44.639,158.767
C07193=1037.289,370.929,368.782,172.955,44.636,158.766
C07194=1037.281,370.683,368.823,172.948,44.632,158.764
C07195=1037.272,370.437,368.863,172.942,44.628,158.763
C07196=1037.264,370.189,368.903,172.935,44.625,158.762
C07197=1037.256,369.942,368.943,172.928,44.622,158.760
C07198=1037.248,369.696,368.983,172.921,44.619,158.759
C07199=1037.240,369.449,369.023,172.914,44.615,158.757
C07200=1037.231,369.203,369.063,172.907,44.612,158.756
C07201=1037.223,368.957,369.103,172.900,44.608,158.754
C07202=1037.215,368.710,369.143,172.894,44.605,158.753
C07203=1037.207,368.462,369.183,172.887,44.602,158.751
C07204=1037.198,368.216,369.222,172.881,44.599,158.750
C07205=1037.190,367.969,369.261,172.874,44.595,158.748
C07206=1037.182,367.723,369.302,172.867,44.592,158.747
C07207=1037.173,367.476,369.341,172.860,44.589,158.745
C07208=1037.166,367.229,369.381,172.853,44.586,158.744
C07209=1037.157,366.983,369.421,172.848,44.582,158.743
C07210=1037.149,366.736,369.461,172.841,44.579,158.741
C07211=1037.141,366.489,369.500,172.834,44.576,158.740
C07212=1037.132,366.243,369.539,172.827,44.573,158.738
C07213=1037.125,365.996,369.579,172.820,44.570,158.737
C07214=1037.116,365.749,369.618,172.814,44.566,158.735
C07215=1037.109,365.502,369.658,172.807,44.563,158.734
C07216=1037.101,365.256,369.697,172.801,44.560,158.733
C07217=1037.093,365.009,369.737,172.794,44.557,158.731
C07218=1037.085,364.762,369.776,172.788,44.554,158.730
C07219=1037.076,364.516,369.815,172.781,44.551,158.728
C07220=1037.069,364.269,369.855,172.774,44.548,158.727
C07221=1037.056,363.891,369.916,172.765,44.543,158.725
C07222=1037.044,363.513,369.975,172.755,44.538,158.723
C07223=1037.032,363.134,370.036,172.745,44.533,158.721
C07224=1037.020,362.756,370.096,172.735,44.528,158.719
C07225=1037.012,362.510,370.135,172.729,44.525,158.717
C07226=1037.004,362.262,370.174,172.722,44.522,158.716
C07227=1036.996,362.015,370.214,172.716,44.519,158.715
C07228=1036.988,361.769,370.252,172.710,44.516,158.713
C07229=1036.981,361.522,370.292,172.703,44.513,158.712
C07230=1036.972,361.275,370.331,172.697,44.510,158.711
C07231=1036.964,361.028,370.370,172.690,44.508,158.709
C07232=1036.956,360.782,370.408,172.685,44.504,158.708
C07233=1036.948,360.534,370.447,172.678,44.501,158.707
C07234=1036.940,360.288,370.486,172.671,44.499,158.705
C07235=1036.932,360.041,370.524,172.666,44.495,158.704
C07236=1036.925,359.794,370.563,172.659,44.493,158.703
C07237=1036.916,359.547,370.603,172.653,44.490,158.701
C07238=1036.909,359.301,370.641,172.647,44.486,158.700
C07239=1036.901,359.053,370.680,172.640,44.484,158.699
C07240=1036.893,358.806,370.718,172.634,44.481,158.698
C07241=1036.885,358.560,370.757,172.628,44.478,158.696
C07242=1036.877,358.313,370.796,172.622,44.475,158.695
C07243=1036.868,358.066,370.834,172.615,44.472,158.694
C07244=1036.861,357.819,370.873,172.610,44.470,158.693
C07245=1036.853,357.572,370.911,172.603,44.467,158.691
C07246=1036.845,357.326,370.950,172.598,44.464,158.690
C07247=1036.837,357.078,370.988,172.591,44.461,158.689
C07248=1036.830,356.832,371.027,172.585,44.458,158.687
C07249=1036.822,356.584,371.066,172.579,44.456,158.686
C07250=1036.814,356.338,371.104,172.573,44.453,158.685
C07251=1036.806,356.091,371.142,172.566,44.450,158.684
C07252=1036.799,355.844,371.181,172.561,44.447,158.682
C07253=1036.791,355.596,371.219,172.554,44.444,158.681
C07254=1036.783,355.350,371.256,172.549,44.442,158.680
C07255=1036.774,355.103,371.295,172.542,44.439,158.679
C07256=1036.767,354.856,371.333,172.537,44.437,158.678
C07257=1036.759,354.609,371.371,172.530,44.434,158.676
C07258=1036.752,354.362,371.409,172.524,44.431,158.675
C07259=1036.743,354.115,371.448,172.518,44.428,158.674
C07260=1036.736,353.868,371.485,172.512,44.425,158.673
C07261=1036.729,353.621,371.524,172.507,44.423,158.672
C07262=1036.720,353.374,371.562,172.500,44.420,158.670
C07263=1036.712,353.127,371.599,172.495,44.417,158.669
C07264=1036.704,352.880,371.638,172.488,44.415,158.668
C07265=1036.697,352.633,371.676,172.483,44.412,158.667
C07266=1036.689,352.386,371.714,172.476,44.410,158.666
C07267=1036.681,352.139,371.752,172.471,44.407,158.664
C07268=1036.674,351.892,371.790,172.465,44.404,158.663
C07269=1036.666,351.646,371.827,172.459,44.402,158.662
C07270=1036.659,351.399,371.865,172.454,44.400,158.661
C07271=1036.651,351.151,371.903,172.448,44.397,158.660
C07272=1036.643,350.904,371.941,172.441,44.394,158.659
C07273=1036.636,350.657,371.978,172.436,44.391,158.657
C07274=1036.628,350.410,372.017,172.430,44.389,158.656
C07275=1036.620,350.163,372.054,172.424,44.387,158.655
C07276=1036.613,349.916,372.092,172.419,44.384,158.654
C07277=1036.601,349.544,372.149,172.409,44.380,158.652
C07278=1036.590,349.171,372.205,172.401,44.376,158.651
C07279=1036.578,348.799,372.262,172.392,44.373,158.649
C07280=1036.567,348.427,372.318,172.384,44.369,158.647
C07281=1036.559,348.180,372.355,172.379,44.366,158.646
C07282=1036.552,347.933,372.393,172.372,44.364,158.645
C07283=1036.543,347.686,372.430,172.367,44.362,158.644
